C05403=1026.650,-101.229,-87.108,166.767,45.129,158.260
C05404=1026.657,-100.943,-87.119,166.771,45.126,158.259
C05405=1026.664,-100.656,-87.129,166.774,45.123,158.259
C05406=1026.670,-100.371,-87.141,166.778,45.121,158.259
C05407=1026.676,-100.120,-87.149,166.781,45.118,158.259
C05408=1026.681,-99.870,-87.160,166.783,45.115,158.259
C05409=1026.687,-99.621,-87.169,166.787,45.113,158.259
C05410=1026.693,-99.371,-87.178,166.789,45.110,158.259
C05411=1026.699,-99.122,-87.188,166.793,45.108,158.259
C05412=1026.705,-98.872,-87.198,166.795,45.105,158.258
C05413=1026.711,-98.622,-87.208,166.799,45.103,158.258
C05414=1026.716,-98.373,-87.217,166.801,45.101,158.258
C05415=1026.722,-98.123,-87.226,166.805,45.098,158.258
C05416=1026.729,-97.873,-87.236,166.807,45.096,158.258
C05417=1026.735,-97.623,-87.246,166.811,45.093,158.258
C05418=1026.740,-97.374,-87.255,166.813,45.091,158.258
C05419=1026.746,-97.124,-87.265,166.817,45.088,158.258
C05420=1026.751,-96.874,-87.275,166.819,45.086,158.257
C05421=1026.757,-96.624,-87.285,166.822,45.084,158.257
C05422=1026.763,-96.374,-87.295,166.825,45.081,158.257
C05423=1026.768,-96.125,-87.304,166.828,45.079,158.257
C05424=1026.774,-95.875,-87.314,166.831,45.077,158.257
C05425=1026.780,-95.625,-87.324,166.834,45.074,158.257
C05426=1026.786,-95.376,-87.335,166.837,45.072,158.257
C05427=1026.792,-95.126,-87.344,166.840,45.069,158.257
C05428=1026.797,-94.876,-87.354,166.843,45.067,158.257
C05429=1026.803,-94.627,-87.364,166.846,45.065,158.257
C05430=1026.808,-94.376,-87.374,166.848,45.062,158.256
C05431=1026.815,-94.127,-87.383,166.852,45.060,158.256
C05432=1026.820,-93.876,-87.393,166.854,45.058,158.256
C05433=1026.826,-93.627,-87.404,166.858,45.055,158.256
C05434=1026.831,-93.378,-87.414,166.860,45.053,158.256
C05435=1026.837,-93.128,-87.423,166.864,45.050,158.256
C05436=1026.843,-92.878,-87.433,166.866,45.048,158.256
C05437=1026.849,-92.628,-87.443,166.869,45.046,158.256
C05438=1026.855,-92.379,-87.454,166.872,45.043,158.255
C05439=1026.861,-92.129,-87.463,166.875,45.041,158.255
C05440=1026.866,-91.879,-87.473,166.878,45.038,158.255
C05441=1026.873,-91.629,-87.483,166.881,45.036,158.255
C05442=1026.878,-91.380,-87.494,166.884,45.033,158.255
C05443=1026.884,-91.130,-87.503,166.887,45.031,158.255
C05444=1026.889,-90.880,-87.513,166.891,45.029,158.255
C05445=1026.896,-90.631,-87.524,166.893,45.026,158.255
C05446=1026.901,-90.381,-87.534,166.895,45.024,158.255
C05447=1026.907,-90.131,-87.543,166.899,45.022,158.254
C05448=1026.913,-89.881,-87.553,166.901,45.020,158.254
C05449=1026.919,-89.632,-87.564,166.905,45.017,158.254
C05450=1026.925,-89.382,-87.574,166.907,45.015,158.254
C05451=1026.931,-89.132,-87.583,166.911,45.012,158.254
C05452=1026.937,-88.883,-87.594,166.913,45.010,158.254
C05453=1026.943,-88.633,-87.604,166.917,45.008,158.254
C05454=1026.948,-88.383,-87.614,166.919,45.005,158.254
C05455=1026.955,-88.133,-87.624,166.922,45.003,158.253
C05456=1026.960,-87.883,-87.634,166.926,45.001,158.253
C05457=1026.967,-87.634,-87.645,166.928,44.998,158.253
C05458=1026.972,-87.384,-87.655,166.932,44.996,158.253
C05459=1026.978,-87.134,-87.665,166.934,44.993,158.253
C05460=1026.984,-86.885,-87.675,166.937,44.991,158.253
C05461=1026.990,-86.635,-87.685,166.940,44.988,158.253
C05462=1026.996,-86.385,-87.696,166.943,44.986,158.253
C05463=1027.001,-86.135,-87.706,166.946,44.984,158.253
C05464=1027.008,-85.886,-87.716,166.948,44.981,158.252
C05465=1027.013,-85.636,-87.726,166.952,44.979,158.252
C05466=1027.019,-85.386,-87.736,166.954,44.976,158.252
C05467=1027.026,-85.103,-87.748,166.958,44.974,158.252
C05468=1027.033,-84.819,-87.760,166.961,44.971,158.252
C05469=1027.040,-84.534,-87.772,166.965,44.968,158.252
C05470=1027.046,-84.250,-87.783,166.968,44.966,158.252
C05471=1027.053,-84.001,-87.793,166.971,44.964,158.251
C05472=1027.058,-83.751,-87.804,166.974,44.961,158.251
C05473=1027.065,-83.502,-87.814,166.977,44.959,158.251
C05474=1027.070,-83.252,-87.824,166.980,44.956,158.251
C05475=1027.077,-83.002,-87.835,166.983,44.954,158.251
C05476=1027.083,-82.752,-87.845,166.986,44.952,158.251
C05477=1027.088,-82.502,-87.856,166.989,44.949,158.251
C05478=1027.094,-82.252,-87.865,166.992,44.947,158.251
C05479=1027.100,-82.003,-87.876,166.995,44.944,158.250
C05480=1027.107,-81.754,-87.886,166.997,44.942,158.250
C05481=1027.112,-81.503,-87.897,167.001,44.939,158.250
C05482=1027.119,-81.254,-87.907,167.003,44.937,158.250
C05483=1027.125,-81.003,-87.917,167.007,44.934,158.250
C05484=1027.130,-80.754,-87.928,167.009,44.932,158.250
C05485=1027.137,-80.505,-87.939,167.013,44.929,158.250
C05486=1027.142,-80.255,-87.949,167.015,44.927,158.250
C05487=1027.149,-80.006,-87.959,167.019,44.925,158.250
C05488=1027.154,-79.756,-87.970,167.021,44.922,158.249
C05489=1027.161,-79.505,-87.980,167.024,44.920,158.249
C05490=1027.166,-79.256,-87.991,167.027,44.918,158.249
C05491=1027.172,-79.006,-88.002,167.030,44.916,158.249
C05492=1027.178,-78.757,-88.012,167.032,44.914,158.249
C05493=1027.184,-78.507,-88.023,167.036,44.911,158.249
C05494=1027.190,-78.257,-88.034,167.038,44.909,158.249
C05495=1027.196,-78.007,-88.045,167.042,44.907,158.249
C05496=1027.202,-77.758,-88.056,167.044,44.905,158.248
C05497=1027.207,-77.508,-88.066,167.047,44.903,158.248
C05498=1027.214,-77.258,-88.076,167.050,44.900,158.248
C05499=1027.220,-77.008,-88.087,167.053,44.898,158.248
C05500=1027.226,-76.759,-88.098,167.056,44.896,158.248
C05501=1027.231,-76.509,-88.109,167.059,44.893,158.248
C05502=1027.237,-76.260,-88.120,167.062,44.891,158.248
C05503=1027.243,-76.010,-88.131,167.065,44.889,158.248
C05504=1027.250,-75.760,-88.141,167.068,44.887,158.248
C05505=1027.255,-75.510,-88.152,167.070,44.884,158.247
C05506=1027.261,-75.261,-88.162,167.074,44.882,158.247
C05507=1027.267,-75.011,-88.173,167.076,44.880,158.247
C05508=1027.273,-74.761,-88.185,167.079,44.877,158.247
C05509=1027.279,-74.512,-88.195,167.082,44.875,158.247
C05510=1027.285,-74.262,-88.206,167.085,44.873,158.247
C05511=1027.290,-74.013,-88.217,167.089,44.871,158.247
C05512=1027.297,-73.763,-88.228,167.091,44.868,158.247
C05513=1027.303,-73.513,-88.239,167.094,44.866,158.247
C05514=1027.308,-73.264,-88.250,167.096,44.864,158.246
C05515=1027.315,-73.013,-88.261,167.100,44.862,158.246
C05516=1027.320,-72.764,-88.272,167.102,44.860,158.246
C05517=1027.326,-72.514,-88.283,167.105,44.858,158.246
C05518=1027.331,-72.265,-88.295,167.109,44.856,158.246
C05519=1027.337,-72.014,-88.306,167.111,44.854,158.246
C05520=1027.343,-71.765,-88.317,167.113,44.851,158.246
C05521=1027.349,-71.515,-88.328,167.117,44.849,158.246
C05522=1027.355,-71.265,-88.339,167.120,44.847,158.246
C05523=1027.361,-71.016,-88.350,167.122,44.845,158.246
C05524=1027.367,-70.766,-88.361,167.125,44.843,158.246
C05525=1027.373,-70.517,-88.373,167.129,44.841,158.246
C05526=1027.378,-70.267,-88.384,167.131,44.839,158.245
C05527=1027.384,-70.017,-88.395,167.134,44.837,158.245
C05528=1027.390,-69.767,-88.406,167.137,44.834,158.245
C05529=1027.396,-69.518,-88.417,167.140,44.832,158.245
C05530=1027.402,-69.268,-88.428,167.142,44.830,158.245
C05531=1027.408,-68.987,-88.441,167.146,44.828,158.245
C05532=1027.416,-68.704,-88.454,167.149,44.825,158.245
///RCONF 1,0,0,1,0,0,0,0,0,0,0,0,0,0,0,0,0,0,0,0,0,0,0,0
C05533=1027.422,-68.423,-88.466,167.152,44.823,158.245
C05534=1027.428,-68.141,-88.479,167.155,44.820,158.245
C05535=1027.435,-67.891,-88.491,167.158,44.818,158.244
C05536=1027.441,-67.641,-88.502,167.161,44.816,158.244
C05537=1027.447,-67.391,-88.513,167.164,44.814,158.244
C05538=1027.453,-67.142,-88.524,167.167,44.812,158.244
C05539=1027.458,-66.892,-88.535,167.170,44.810,158.244
C05540=1027.464,-66.642,-88.547,167.173,44.807,158.244
C05541=1027.470,-66.393,-88.558,167.175,44.805,158.244
C05542=1027.476,-66.143,-88.570,167.178,44.803,158.244
C05543=1027.482,-65.894,-88.581,167.181,44.801,158.244
C05544=1027.488,-65.644,-88.592,167.184,44.799,158.244
C05545=1027.494,-65.394,-88.604,167.187,44.797,158.244
C05546=1027.499,-65.144,-88.615,167.190,44.794,158.243
C05547=1027.506,-64.895,-88.627,167.193,44.792,158.243
C05548=1027.512,-64.645,-88.638,167.195,44.790,158.243
C05549=1027.518,-64.395,-88.649,167.199,44.788,158.243
C05550=1027.524,-64.146,-88.660,167.201,44.786,158.243
C05551=1027.530,-63.896,-88.672,167.204,44.784,158.243
C05552=1027.536,-63.646,-88.683,167.206,44.781,158.243
C05553=1027.542,-63.397,-88.695,167.210,44.779,158.243
C05554=1027.548,-63.147,-88.706,167.213,44.777,158.243
C05555=1027.555,-62.898,-88.718,167.215,44.775,158.242
C05556=1027.560,-62.648,-88.729,167.219,44.773,158.242
C05557=1027.566,-62.398,-88.741,167.221,44.770,158.242
C05558=1027.572,-62.149,-88.752,167.224,44.768,158.242
C05559=1027.578,-61.899,-88.763,167.227,44.766,158.242
C05560=1027.584,-61.650,-88.775,167.230,44.764,158.242
C05561=1027.590,-61.399,-88.787,167.233,44.762,158.242
C05562=1027.596,-61.150,-88.798,167.235,44.760,158.242
C05563=1027.602,-60.900,-88.810,167.239,44.757,158.242
C05564=1027.608,-60.651,-88.821,167.241,44.755,158.241
C05565=1027.615,-60.401,-88.833,167.244,44.753,158.241
C05566=1027.620,-60.151,-88.844,167.247,44.751,158.241
C05567=1027.626,-59.902,-88.856,167.250,44.749,158.241
C05568=1027.633,-59.652,-88.867,167.252,44.747,158.241
C05569=1027.639,-59.403,-88.879,167.255,44.745,158.241
C05570=1027.645,-59.152,-88.890,167.259,44.742,158.241
C05571=1027.650,-58.903,-88.902,167.261,44.740,158.241
C05572=1027.657,-58.653,-88.914,167.264,44.738,158.241
C05573=1027.663,-58.404,-88.925,167.267,44.736,158.240
C05574=1027.669,-58.154,-88.936,167.270,44.734,158.240
C05575=1027.676,-57.904,-88.948,167.272,44.732,158.240
C05576=1027.681,-57.655,-88.960,167.276,44.729,158.240
C05577=1027.687,-57.405,-88.972,167.278,44.727,158.240
C05578=1027.694,-57.155,-88.983,167.281,44.725,158.240
C05579=1027.700,-56.906,-88.995,167.284,44.723,158.240
C05580=1027.706,-56.656,-89.007,167.287,44.721,158.240
C05581=1027.712,-56.407,-89.018,167.289,44.718,158.240
C05582=1027.718,-56.157,-89.030,167.292,44.716,158.239
C05583=1027.725,-55.907,-89.041,167.296,44.714,158.239
C05584=1027.731,-55.658,-89.053,167.298,44.712,158.239
C05585=1027.736,-55.408,-89.065,167.301,44.709,158.239
C05586=1027.743,-55.158,-89.077,167.303,44.707,158.239
C05587=1027.749,-54.909,-89.088,167.307,44.705,158.239
C05588=1027.756,-54.660,-89.100,167.309,44.703,158.239
C05589=1027.761,-54.409,-89.112,167.312,44.700,158.239
C05590=1027.768,-54.159,-89.124,167.315,44.698,158.239
C05591=1027.774,-53.911,-89.136,167.318,44.696,158.238
C05592=1027.780,-53.660,-89.147,167.321,44.694,158.238
C05593=1027.786,-53.410,-89.159,167.324,44.692,158.238
C05594=1027.792,-53.162,-89.171,167.327,44.690,158.238
C05595=1027.799,-52.881,-89.184,167.329,44.687,158.238
C05596=1027.806,-52.600,-89.198,167.333,44.685,158.238
C05597=1027.813,-52.319,-89.210,167.336,44.682,158.238
C05598=1027.821,-52.038,-89.224,167.340,44.680,158.238
C05599=1027.826,-51.788,-89.236,167.342,44.678,158.237
C05600=1027.832,-51.539,-89.247,167.345,44.675,158.237
C05601=1027.839,-51.290,-89.259,167.347,44.673,158.237
C05602=1027.846,-51.040,-89.271,167.351,44.671,158.237
C05603=1027.851,-50.789,-89.283,167.353,44.668,158.237
C05604=1027.858,-50.540,-89.295,167.356,44.666,158.237
C05605=1027.863,-50.291,-89.307,167.358,44.664,158.237
C05606=1027.869,-50.041,-89.320,167.362,44.662,158.237
C05607=1027.876,-49.791,-89.332,167.365,44.660,158.236
C05608=1027.882,-49.541,-89.344,167.367,44.658,158.236
C05609=1027.888,-49.293,-89.356,167.370,44.656,158.236
C05610=1027.894,-49.043,-89.369,167.372,44.654,158.236
C05611=1027.900,-48.793,-89.381,167.376,44.652,158.236
C05612=1027.906,-48.543,-89.393,167.379,44.650,158.236
C05613=1027.912,-48.294,-89.405,167.381,44.648,158.236
C05614=1027.917,-48.044,-89.418,167.384,44.646,158.236
C05615=1027.924,-47.795,-89.430,167.386,44.644,158.236
C05616=1027.930,-47.545,-89.442,167.389,44.642,158.236
C05617=1027.937,-47.295,-89.454,167.393,44.640,158.236
C05618=1027.942,-47.046,-89.466,167.395,44.638,158.235
C05619=1027.948,-46.796,-89.479,167.398,44.636,158.235
C05620=1027.954,-46.546,-89.491,167.400,44.634,158.235
C05621=1027.960,-46.297,-89.503,167.403,44.632,158.235
C05622=1027.966,-46.047,-89.516,167.407,44.630,158.235
C05623=1027.972,-45.798,-89.528,167.409,44.628,158.235
C05624=1027.978,-45.548,-89.540,167.412,44.626,158.235
C05625=1027.984,-45.298,-89.553,167.414,44.624,158.235
C05626=1027.991,-45.048,-89.565,167.417,44.622,158.235
C05627=1027.997,-44.799,-89.577,167.420,44.619,158.235
C05628=1028.003,-44.549,-89.590,167.423,44.617,158.234
C05629=1028.009,-44.300,-89.601,167.426,44.615,158.234
C05630=1028.015,-44.050,-89.614,167.428,44.614,158.234
C05631=1028.020,-43.800,-89.627,167.431,44.612,158.234
C05632=1028.027,-43.551,-89.639,167.433,44.610,158.234
C05633=1028.033,-43.301,-89.652,167.437,44.607,158.234
C05634=1028.039,-43.051,-89.664,167.440,44.605,158.234
C05635=1028.046,-42.802,-89.676,167.442,44.604,158.234
C05636=1028.052,-42.552,-89.689,167.445,44.602,158.234
C05637=1028.058,-42.302,-89.701,167.447,44.600,158.234
C05638=1028.064,-42.052,-89.713,167.451,44.597,158.233
C05639=1028.070,-41.804,-89.726,167.453,44.595,158.233
C05640=1028.076,-41.554,-89.739,167.456,44.593,158.233
C05641=1028.083,-41.304,-89.751,167.459,44.591,158.233
C05642=1028.088,-41.055,-89.763,167.461,44.589,158.233
C05643=1028.094,-40.805,-89.776,167.464,44.587,158.233
C05644=1028.101,-40.556,-89.789,167.467,44.585,158.233
C05645=1028.107,-40.306,-89.801,167.470,44.583,158.233
C05646=1028.113,-40.056,-89.814,167.473,44.581,158.233
C05647=1028.120,-39.806,-89.826,167.475,44.579,158.232
C05648=1028.126,-39.557,-89.839,167.478,44.576,158.232
C05649=1028.132,-39.307,-89.851,167.481,44.574,158.232
C05650=1028.139,-39.058,-89.863,167.484,44.572,158.232
C05651=1028.144,-38.808,-89.876,167.486,44.570,158.232
C05652=1028.151,-38.558,-89.889,167.489,44.568,158.232
C05653=1028.157,-38.309,-89.902,167.492,44.566,158.232
C05654=1028.162,-38.059,-89.914,167.494,44.564,158.232
C05655=1028.169,-37.809,-89.928,167.497,44.562,158.232
C05656=1028.175,-37.560,-89.940,167.499,44.560,158.231
C05657=1028.181,-37.310,-89.953,167.503,44.558,158.231
C05658=1028.187,-37.060,-89.966,167.506,44.557,158.231
C05659=1028.194,-36.780,-89.981,167.508,44.554,158.231
C05660=1028.200,-36.500,-89.994,167.512,44.552,158.231
C05661=1028.207,-36.220,-90.009,167.514,44.550,158.231
C05662=1028.214,-35.940,-90.023,167.518,44.548,158.231
C05663=1028.220,-35.690,-90.037,167.521,44.546,158.231
C05664=1028.226,-35.440,-90.049,167.523,44.544,158.231
C05665=1028.232,-35.191,-90.062,167.526,44.542,158.231
C05666=1028.238,-34.941,-90.075,167.528,44.540,158.231
C05667=1028.244,-34.691,-90.087,167.531,44.538,158.230
C05668=1028.250,-34.442,-90.101,167.534,44.536,158.230
C05669=1028.257,-34.193,-90.113,167.536,44.534,158.230
C05670=1028.263,-33.943,-90.126,167.539,44.532,158.230
C05671=1028.269,-33.693,-90.139,167.542,44.530,158.230
C05672=1028.276,-33.443,-90.152,167.545,44.528,158.230
C05673=1028.282,-33.194,-90.165,167.548,44.526,158.230
C05674=1028.288,-32.944,-90.178,167.550,44.524,158.230
C05675=1028.294,-32.695,-90.191,167.553,44.522,158.230
C05676=1028.300,-32.445,-90.204,167.555,44.520,158.230
C05677=1028.306,-32.196,-90.217,167.558,44.519,158.229
C05678=1028.312,-31.946,-90.230,167.561,44.517,158.229
C05679=1028.318,-31.697,-90.243,167.563,44.515,158.229
C05680=1028.324,-31.447,-90.255,167.567,44.512,158.229
C05681=1028.330,-31.198,-90.269,167.570,44.511,158.229
C05682=1028.337,-30.948,-90.282,167.572,44.509,158.229
C05683=1028.343,-30.698,-90.295,167.575,44.507,158.229
C05684=1028.349,-30.448,-90.308,167.577,44.505,158.229
C05685=1028.356,-30.199,-90.321,167.580,44.502,158.228
C05686=1028.361,-29.949,-90.334,167.582,44.500,158.228
C05687=1028.368,-29.700,-90.347,167.585,44.498,158.228
C05688=1028.374,-29.450,-90.360,167.587,44.496,158.228
///RCONF 1,0,0,0,0,0,0,0,0,0,0,0,0,0,0,0,0,0,0,0,0,0,0,0
C05689=1028.380,-29.201,-90.373,167.591,44.494,158.228
C05690=1028.387,-28.951,-90.387,167.594,44.492,158.228
C05691=1028.393,-28.701,-90.399,167.596,44.490,158.228
C05692=1028.399,-28.452,-90.413,167.599,44.488,158.228
C05693=1028.405,-28.203,-90.426,167.602,44.486,158.228
C05694=1028.411,-27.953,-90.438,167.604,44.484,158.228
C05695=1028.418,-27.703,-90.452,167.607,44.482,158.227
C05696=1028.424,-27.453,-90.465,167.609,44.480,158.227
C05697=1028.430,-27.204,-90.479,167.612,44.478,158.227
C05698=1028.436,-26.954,-90.491,167.615,44.476,158.227
C05699=1028.442,-26.705,-90.504,167.617,44.475,158.227
C05700=1028.448,-26.456,-90.518,167.620,44.473,158.227
C05701=1028.455,-26.205,-90.532,167.623,44.470,158.227
C05702=1028.461,-25.956,-90.545,167.626,44.468,158.227
C05703=1028.467,-25.707,-90.558,167.629,44.467,158.227
C05704=1028.473,-25.457,-90.571,167.631,44.465,158.227
C05705=1028.478,-25.207,-90.585,167.634,44.463,158.227
C05706=1028.485,-24.958,-90.598,167.637,44.461,158.226
C05707=1028.491,-24.708,-90.612,167.639,44.459,158.226
C05708=1028.498,-24.459,-90.625,167.642,44.457,158.226
C05709=1028.503,-24.209,-90.639,167.644,44.456,158.226
C05710=1028.509,-23.960,-90.652,167.647,44.454,158.226
C05711=1028.516,-23.710,-90.666,167.650,44.452,158.226
C05712=1028.522,-23.460,-90.678,167.652,44.450,158.226
C05713=1028.527,-23.211,-90.692,167.655,44.448,158.226
C05714=1028.534,-22.961,-90.705,167.657,44.446,158.226
C05715=1028.540,-22.718,-90.719,167.660,44.445,158.226
C05716=1028.546,-22.474,-90.732,167.663,44.443,158.226
C05717=1028.552,-22.230,-90.745,167.665,44.441,158.225
C05718=1028.558,-21.987,-90.759,167.668,44.439,158.225
C05719=1028.564,-21.743,-90.772,167.671,44.437,158.225
C05720=1028.570,-21.499,-90.785,167.673,44.435,158.225
C05721=1028.576,-21.255,-90.799,167.676,44.433,158.225
C05722=1028.582,-21.011,-90.811,167.678,44.431,158.225
C05723=1028.590,-20.718,-90.827,167.681,44.429,158.225
C05724=1028.597,-20.426,-90.843,167.685,44.427,158.225
C05725=1028.605,-20.133,-90.859,167.687,44.424,158.224
C05726=1028.611,-19.841,-90.875,167.691,44.422,158.224
C05727=1028.618,-19.591,-90.889,167.693,44.420,158.224
C05728=1028.624,-19.341,-90.902,167.696,44.418,158.224
C05729=1028.630,-19.092,-90.916,167.698,44.416,158.224
C05730=1028.637,-18.842,-90.930,167.701,44.414,158.224
C05731=1028.643,-18.593,-90.943,167.704,44.412,158.224
C05732=1028.648,-18.343,-90.957,167.706,44.410,158.224
C05733=1028.655,-18.093,-90.970,167.709,44.408,158.224
C05734=1028.661,-17.844,-90.984,167.711,44.406,158.223
C05735=1028.668,-17.594,-90.997,167.714,44.405,158.223
C05736=1028.674,-17.344,-91.011,167.717,44.403,158.223
C05737=1028.680,-17.095,-91.024,167.719,44.401,158.223
C05738=1028.686,-16.846,-91.038,167.722,44.399,158.223
C05739=1028.692,-16.596,-91.053,167.724,44.397,158.223
C05740=1028.699,-16.347,-91.066,167.727,44.395,158.223
C05741=1028.705,-16.097,-91.080,167.730,44.393,158.223
C05742=1028.711,-15.847,-91.093,167.732,44.391,158.223
C05743=1028.717,-15.598,-91.107,167.735,44.389,158.222
C05744=1028.724,-15.348,-91.120,167.737,44.387,158.222
C05745=1028.730,-15.099,-91.135,167.740,44.385,158.222
C05746=1028.737,-14.849,-91.149,167.743,44.384,158.222
C05747=1028.742,-14.599,-91.162,167.746,44.382,158.222
C05748=1028.747,-14.350,-91.176,167.748,44.380,158.222
C05749=1028.755,-14.101,-91.191,167.751,44.378,158.222
C05750=1028.760,-13.851,-91.204,167.753,44.376,158.222
C05751=1028.767,-13.601,-91.218,167.756,44.374,158.222
C05752=1028.772,-13.351,-91.232,167.759,44.372,158.222
C05753=1028.779,-13.103,-91.246,167.761,44.370,158.221
C05754=1028.785,-12.853,-91.260,167.764,44.369,158.222
C05755=1028.791,-12.603,-91.273,167.767,44.367,158.221
C05756=1028.798,-12.354,-91.288,167.769,44.365,158.221
C05757=1028.803,-12.104,-91.302,167.772,44.363,158.221
C05758=1028.810,-11.854,-91.316,167.774,44.361,158.221
C05759=1028.816,-11.605,-91.330,167.777,44.359,158.221
C05760=1028.822,-11.356,-91.344,167.780,44.357,158.221
C05761=1028.828,-11.106,-91.359,167.782,44.355,158.221
C05762=1028.834,-10.857,-91.372,167.785,44.353,158.221
C05763=1028.841,-10.607,-91.386,167.788,44.352,158.221
C05764=1028.847,-10.358,-91.400,167.790,44.350,158.221
C05765=1028.853,-10.108,-91.414,167.793,44.348,158.220
C05766=1028.859,-9.858,-91.428,167.795,44.346,158.220
C05767=1028.866,-9.609,-91.443,167.798,44.344,158.220
C05768=1028.871,-9.359,-91.456,167.801,44.343,158.220
C05769=1028.878,-9.110,-91.471,167.803,44.341,158.220
C05770=1028.884,-8.860,-91.485,167.806,44.339,158.220
C05771=1028.891,-8.611,-91.499,167.808,44.337,158.220
C05772=1028.896,-8.361,-91.513,167.811,44.335,158.220
C05773=1028.903,-8.112,-91.528,167.813,44.333,158.219
C05774=1028.909,-7.862,-91.541,167.815,44.331,158.219
C05775=1028.915,-7.612,-91.555,167.818,44.329,158.219
C05776=1028.922,-7.364,-91.569,167.821,44.328,158.219
C05777=1028.928,-7.113,-91.584,167.823,44.326,158.219
C05778=1028.933,-6.864,-91.598,167.826,44.324,158.219
C05779=1028.940,-6.614,-91.612,167.828,44.322,158.219
C05780=1028.947,-6.365,-91.627,167.831,44.320,158.219
C05781=1028.953,-6.115,-91.640,167.834,44.318,158.219
C05782=1028.959,-5.866,-91.655,167.836,44.316,158.219
C05783=1028.965,-5.616,-91.669,167.839,44.314,158.218
C05784=1028.972,-5.367,-91.683,167.841,44.312,158.218
C05785=1028.978,-5.118,-91.698,167.844,44.310,158.218
C05786=1028.984,-4.868,-91.711,167.847,44.309,158.218
C05787=1028.991,-4.585,-91.727,167.849,44.307,158.218
C05788=1028.998,-4.302,-91.744,167.853,44.304,158.218
C05789=1029.006,-4.020,-91.760,167.855,44.302,158.218
C05790=1029.013,-3.736,-91.776,167.858,44.300,158.218
C05791=1029.018,-3.487,-91.791,167.861,44.298,158.217
C05792=1029.025,-3.238,-91.806,167.863,44.297,158.217
C05793=1029.031,-2.988,-91.821,167.866,44.295,158.217
C05794=1029.037,-2.739,-91.835,167.869,44.293,158.217
C05795=1029.043,-2.489,-91.849,167.871,44.291,158.217
C05796=1029.049,-2.240,-91.864,167.874,44.289,158.217
C05797=1029.056,-1.991,-91.878,167.877,44.288,158.217
C05798=1029.061,-1.741,-91.892,167.878,44.286,158.217
C05799=1029.068,-1.491,-91.907,167.881,44.284,158.217
C05800=1029.074,-1.242,-91.922,167.883,44.282,158.217
C05801=1029.080,-0.993,-91.937,167.886,44.281,158.217
C05802=1029.086,-0.742,-91.951,167.889,44.279,158.216
C05803=1029.092,-0.494,-91.966,167.891,44.277,158.216
C05804=1029.098,-0.244,-91.980,167.894,44.275,158.216
C05805=1029.105,0.006,-91.995,167.897,44.273,158.216
C05806=1029.110,0.255,-92.010,167.898,44.271,158.216
C05807=1029.116,0.505,-92.024,167.901,44.270,158.216
C05808=1029.123,0.755,-92.039,167.904,44.268,158.216
C05809=1029.129,1.004,-92.054,167.906,44.266,158.216
C05810=1029.135,1.253,-92.069,167.909,44.264,158.216
C05811=1029.141,1.503,-92.084,167.911,44.262,158.216
C05812=1029.147,1.752,-92.098,167.914,44.261,158.216
C05813=1029.153,2.002,-92.112,167.917,44.259,158.215
C05814=1029.160,2.252,-92.127,167.918,44.258,158.215
C05815=1029.166,2.500,-92.141,167.921,44.256,158.215
C05816=1029.173,2.750,-92.156,167.924,44.254,158.215
C05817=1029.179,3.000,-92.171,167.926,44.252,158.215
C05818=1029.185,3.249,-92.186,167.929,44.251,158.215
C05819=1029.191,3.498,-92.201,167.932,44.249,158.215
C05820=1029.197,3.748,-92.216,167.934,44.247,158.215
C05821=1029.203,3.997,-92.230,167.937,44.245,158.215
C05822=1029.210,4.247,-92.245,167.939,44.243,158.214
C05823=1029.216,4.496,-92.260,167.941,44.241,158.214
C05824=1029.221,4.746,-92.274,167.944,44.239,158.214
C05825=1029.228,4.996,-92.289,167.947,44.238,158.214
C05826=1029.234,5.245,-92.304,167.949,44.236,158.214
C05827=1029.241,5.495,-92.319,167.952,44.234,158.214
C05828=1029.246,5.744,-92.334,167.954,44.232,158.214
C05829=1029.253,5.993,-92.348,167.957,44.230,158.214
C05830=1029.259,6.243,-92.363,167.960,44.228,158.214
C05831=1029.266,6.493,-92.378,167.961,44.227,158.213
C05832=1029.271,6.742,-92.393,167.964,44.225,158.213
C05833=1029.278,6.991,-92.408,167.966,44.223,158.213
C05834=1029.284,7.241,-92.423,167.969,44.221,158.213
C05835=1029.290,7.491,-92.438,167.972,44.220,158.213
C05836=1029.297,7.740,-92.453,167.974,44.218,158.213
C05837=1029.303,7.989,-92.467,167.977,44.216,158.213
C05838=1029.309,8.239,-92.482,167.980,44.214,158.213
C05839=1029.315,8.489,-92.497,167.981,44.212,158.213
C05840=1029.322,8.738,-92.513,167.984,44.210,158.212
C05841=1029.328,8.987,-92.528,167.986,44.208,158.212
C05842=1029.334,9.236,-92.542,167.989,44.206,158.212
C05843=1029.341,9.486,-92.557,167.992,44.204,158.212
C05844=1029.347,9.736,-92.572,167.994,44.202,158.212
C05845=1029.353,9.985,-92.587,167.997,44.200,158.212
C05846=1029.360,10.235,-92.602,167.999,44.199,158.212
C05847=1029.366,10.484,-92.617,168.002,44.197,158.212
C05848=1029.372,10.734,-92.632,168.004,44.196,158.212
C05849=1029.378,10.983,-92.647,168.006,44.194,158.211
C05850=1029.385,11.232,-92.662,168.009,44.192,158.211
C05851=1029.392,11.517,-92.679,168.011,44.189,158.211
C05852=1029.399,11.802,-92.696,168.015,44.187,158.211
C05853=1029.407,12.087,-92.713,168.018,44.185,158.211
C05854=1029.414,12.371,-92.731,168.020,44.183,158.211
C05855=1029.420,12.621,-92.746,168.023,44.181,158.211
C05856=1029.427,12.871,-92.760,168.025,44.179,158.210
C05857=1029.433,13.120,-92.775,168.028,44.177,158.210
C05858=1029.440,13.369,-92.791,168.031,44.175,158.210
C05859=1029.445,13.618,-92.806,168.033,44.174,158.210
C05860=1029.452,13.868,-92.821,168.036,44.172,158.210
C05861=1029.458,14.118,-92.836,168.037,44.170,158.210
C05862=1029.464,14.367,-92.852,168.040,44.168,158.210
C05863=1029.471,14.617,-92.867,168.043,44.166,158.210
C05864=1029.477,14.866,-92.882,168.046,44.165,158.210
C05865=1029.484,15.115,-92.897,168.048,44.163,158.209
C05866=1029.489,15.365,-92.913,168.051,44.161,158.209
C05867=1029.496,15.615,-92.928,168.052,44.159,158.209
C05868=1029.502,15.863,-92.943,168.055,44.157,158.209
C05869=1029.508,16.113,-92.958,168.058,44.155,158.209
C05870=1029.514,16.363,-92.974,168.060,44.154,158.209
C05871=1029.520,16.612,-92.989,168.063,44.152,158.209
C05872=1029.527,16.862,-93.004,168.065,44.151,158.209
C05873=1029.532,17.112,-93.020,168.067,44.149,158.209
C05874=1029.539,17.361,-93.035,168.070,44.147,158.208
C05875=1029.546,17.610,-93.050,168.072,44.145,158.208
C05876=1029.552,17.859,-93.066,168.075,44.143,158.208
C05877=1029.558,18.109,-93.082,168.078,44.142,158.208
C05878=1029.564,18.359,-93.097,168.079,44.140,158.208
C05879=1029.571,18.608,-93.112,168.082,44.138,158.208
C05880=1029.577,18.858,-93.128,168.085,44.136,158.208
C05881=1029.583,19.107,-93.143,168.087,44.134,158.208
C05882=1029.589,19.356,-93.158,168.090,44.132,158.208
C05883=1029.596,19.605,-93.174,168.091,44.130,158.207
C05884=1029.601,19.855,-93.189,168.094,44.129,158.207
C05885=1029.608,20.104,-93.205,168.097,44.127,158.207
C05886=1029.614,20.354,-93.220,168.099,44.125,158.207
C05887=1029.620,20.603,-93.236,168.102,44.123,158.207
C05888=1029.626,20.853,-93.252,168.104,44.122,158.207
C05889=1029.633,21.102,-93.267,168.106,44.121,158.207
C05890=1029.639,21.352,-93.282,168.109,44.119,158.207
C05891=1029.645,21.601,-93.298,168.112,44.117,158.207
C05892=1029.651,21.851,-93.313,168.114,44.115,158.206
C05893=1029.657,22.100,-93.330,168.116,44.113,158.206
C05894=1029.664,22.350,-93.345,168.119,44.111,158.206
C05895=1029.670,22.599,-93.361,168.121,44.110,158.206
C05896=1029.676,22.848,-93.377,168.124,44.108,158.206
C05897=1029.682,23.098,-93.392,168.127,44.106,158.206
C05898=1029.689,23.347,-93.408,168.128,44.104,158.206
C05899=1029.695,23.597,-93.423,168.131,44.102,158.206
C05900=1029.701,23.846,-93.439,168.133,44.100,158.206
C05901=1029.708,24.095,-93.455,168.136,44.099,158.206
C05902=1029.713,24.345,-93.470,168.139,44.097,158.205
C05903=1029.720,24.594,-93.486,168.140,44.096,158.205
C05904=1029.726,24.843,-93.502,168.143,44.094,158.205
C05905=1029.732,25.093,-93.517,168.146,44.092,158.205
C05906=1029.739,25.343,-93.534,168.148,44.090,158.205
C05907=1029.746,25.592,-93.549,168.151,44.088,158.205
C05908=1029.752,25.842,-93.564,168.152,44.086,158.205
C05909=1029.758,26.091,-93.580,168.155,44.085,158.205
C05910=1029.765,26.340,-93.596,168.158,44.083,158.204
C05911=1029.770,26.590,-93.612,168.160,44.081,158.204
C05912=1029.777,26.839,-93.627,168.162,44.079,158.204
C05913=1029.783,27.089,-93.644,168.165,44.078,158.204
C05914=1029.789,27.338,-93.660,168.167,44.076,158.204
C05915=1029.797,27.624,-93.677,168.170,44.074,158.204
C05916=1029.804,27.910,-93.695,168.172,44.072,158.204
C05917=1029.811,28.196,-93.714,168.176,44.070,158.204
C05918=1029.818,28.482,-93.732,168.179,44.068,158.203
C05919=1029.823,28.732,-93.748,168.181,44.066,158.203
C05920=1029.830,28.981,-93.764,168.183,44.064,158.203
C05921=1029.836,29.230,-93.780,168.186,44.063,158.203
C05922=1029.842,29.479,-93.796,168.188,44.061,158.203
C05923=1029.849,29.729,-93.812,168.191,44.059,158.203
C05924=1029.855,29.979,-93.828,168.193,44.057,158.203
C05925=1029.861,30.228,-93.845,168.195,44.056,158.203
C05926=1029.868,30.478,-93.860,168.198,44.054,158.203
C05927=1029.874,30.727,-93.876,168.201,44.052,158.202
C05928=1029.879,30.976,-93.892,168.202,44.051,158.202
C05929=1029.886,31.225,-93.908,168.205,44.049,158.202
C05930=1029.892,31.475,-93.924,168.208,44.047,158.202
C05931=1029.899,31.725,-93.941,168.210,44.046,158.202
C05932=1029.905,31.974,-93.956,168.212,44.044,158.202
C05933=1029.911,32.223,-93.973,168.214,44.042,158.202
C05934=1029.917,32.472,-93.989,168.217,44.040,158.202
C05935=1029.923,32.722,-94.005,168.220,44.039,158.202
C05936=1029.930,32.971,-94.021,168.221,44.037,158.201
C05937=1029.936,33.221,-94.036,168.224,44.035,158.201
C05938=1029.942,33.471,-94.053,168.227,44.033,158.201
C05939=1029.949,33.720,-94.069,168.229,44.031,158.201
C05940=1029.955,33.969,-94.085,168.231,44.030,158.201
C05941=1029.961,34.219,-94.101,168.234,44.028,158.201
C05942=1029.967,34.468,-94.117,168.236,44.026,158.201
C05943=1029.973,34.717,-94.133,168.239,44.025,158.201
C05944=1029.980,34.967,-94.150,168.240,44.023,158.201
C05945=1029.986,35.216,-94.166,168.243,44.021,158.200
C05946=1029.993,35.465,-94.182,168.246,44.019,158.200
C05947=1029.998,35.715,-94.198,168.248,44.017,158.200
C05948=1030.005,35.965,-94.214,168.250,44.016,158.200
C05949=1030.012,36.214,-94.230,168.253,44.014,158.200
C05950=1030.018,36.463,-94.246,168.255,44.012,158.200
C05951=1030.024,36.712,-94.263,168.258,44.010,158.200
C05952=1030.030,36.961,-94.280,168.260,44.009,158.200
C05953=1030.037,37.211,-94.296,168.262,44.007,158.199
C05954=1030.043,37.460,-94.312,168.265,44.006,158.199
C05955=1030.049,37.710,-94.328,168.268,44.004,158.199
C05956=1030.055,37.959,-94.344,168.269,44.002,158.199
C05957=1030.062,38.209,-94.361,168.272,44.000,158.199
C05958=1030.068,38.458,-94.377,168.275,43.999,158.199
C05959=1030.074,38.707,-94.394,168.276,43.997,158.199
C05960=1030.080,38.956,-94.410,168.279,43.995,158.199
C05961=1030.086,39.206,-94.427,168.281,43.993,158.199
C05962=1030.092,39.456,-94.443,168.284,43.992,158.199
C05963=1030.098,39.705,-94.460,168.286,43.990,158.198
C05964=1030.104,39.955,-94.476,168.288,43.988,158.198
C05965=1030.110,40.203,-94.493,168.291,43.986,158.198
C05966=1030.117,40.453,-94.509,168.294,43.985,158.198
C05967=1030.123,40.703,-94.526,168.295,43.984,158.198
C05968=1030.129,40.952,-94.542,168.298,43.982,158.198
C05969=1030.135,41.201,-94.559,168.301,43.980,158.198
C05970=1030.142,41.451,-94.576,168.302,43.978,158.198
C05971=1030.148,41.700,-94.592,168.305,43.977,158.198
C05972=1030.154,41.950,-94.608,168.308,43.975,158.197
C05973=1030.161,42.199,-94.625,168.310,43.973,158.197
C05974=1030.167,42.448,-94.641,168.312,43.971,158.197
C05975=1030.173,42.697,-94.657,168.315,43.969,158.197
C05976=1030.179,42.946,-94.674,168.317,43.968,158.197
C05977=1030.185,43.196,-94.692,168.319,43.966,158.197
C05978=1030.191,43.446,-94.708,168.322,43.965,158.197
C05979=1030.199,43.731,-94.727,168.324,43.963,158.197
C05980=1030.205,44.018,-94.746,168.327,43.961,158.197
C05981=1030.212,44.303,-94.766,168.330,43.959,158.196
C05982=1030.219,44.589,-94.785,168.332,43.958,158.196
C05983=1030.225,44.838,-94.802,168.335,43.956,158.196
C05984=1030.231,45.089,-94.819,168.337,43.954,158.196
C05985=1030.237,45.338,-94.835,168.339,43.953,158.196
C05986=1030.243,45.587,-94.852,168.342,43.951,158.196
C05987=1030.250,45.837,-94.869,168.344,43.949,158.196
C05988=1030.256,46.086,-94.886,168.346,43.948,158.196
C05989=1030.262,46.335,-94.902,168.349,43.946,158.196
C05990=1030.268,46.584,-94.920,168.352,43.944,158.195
C05991=1030.274,46.834,-94.936,168.353,43.943,158.195
C05992=1030.281,47.083,-94.953,168.356,43.941,158.195
C05993=1030.286,47.333,-94.970,168.359,43.939,158.195
C05994=1030.293,47.582,-94.987,168.360,43.938,158.195
C05995=1030.299,47.831,-95.003,168.363,43.936,158.195
C05996=1030.305,48.080,-95.021,168.366,43.934,158.195
C05997=1030.311,48.330,-95.038,168.367,43.933,158.195
C05998=1030.317,48.579,-95.055,168.370,43.931,158.195
C05999=1030.323,48.829,-95.071,168.373,43.930,158.195
C06000=1030.330,49.078,-95.088,168.374,43.928,158.194
C06001=1030.335,49.327,-95.105,168.377,43.927,158.194
C06002=1030.342,49.577,-95.122,168.380,43.925,158.194
C06003=1030.348,49.826,-95.139,168.381,43.923,158.194
C06004=1030.355,50.075,-95.156,168.384,43.922,158.194
C06005=1030.360,50.324,-95.174,168.387,43.920,158.194
C06006=1030.366,50.574,-95.190,168.389,43.918,158.194
C06007=1030.373,50.823,-95.207,168.391,43.916,158.194
C06008=1030.379,51.073,-95.223,168.394,43.915,158.194
C06009=1030.385,51.322,-95.241,168.396,43.913,158.194
C06010=1030.391,51.571,-95.258,168.398,43.911,158.193
C06011=1030.397,51.820,-95.275,168.401,43.910,158.193
C06012=1030.404,52.070,-95.292,168.403,43.908,158.193
C06013=1030.409,52.320,-95.309,168.405,43.907,158.193
C06014=1030.416,52.569,-95.326,168.408,43.905,158.193
C06015=1030.422,52.818,-95.343,168.410,43.903,158.193
C06016=1030.429,53.068,-95.360,168.412,43.902,158.193
C06017=1030.434,53.317,-95.377,168.415,43.900,158.193
C06018=1030.441,53.565,-95.394,168.417,43.898,158.192
C06019=1030.447,53.816,-95.411,168.420,43.896,158.192
C06020=1030.453,54.065,-95.428,168.421,43.894,158.192
C06021=1030.460,54.314,-95.446,168.424,43.893,158.192
C06022=1030.466,54.563,-95.462,168.427,43.891,158.192
C06023=1030.472,54.813,-95.479,168.428,43.890,158.192
C06024=1030.478,55.062,-95.497,168.431,43.888,158.192
C06025=1030.485,55.311,-95.514,168.434,43.886,158.192
C06026=1030.491,55.561,-95.531,168.435,43.885,158.192
C06027=1030.498,55.810,-95.548,168.438,43.883,158.191
C06028=1030.503,56.059,-95.565,168.441,43.881,158.191
C06029=1030.510,56.309,-95.582,168.443,43.879,158.191
C06030=1030.516,56.558,-95.599,168.445,43.877,158.191
C06031=1030.522,56.808,-95.617,168.448,43.876,158.191
C06032=1030.528,57.056,-95.634,168.450,43.874,158.191
C06033=1030.535,57.306,-95.651,168.452,43.873,158.191
C06034=1030.541,57.555,-95.668,168.455,43.871,158.190
C06035=1030.547,57.805,-95.685,168.457,43.869,158.190
C06036=1030.554,58.054,-95.702,168.460,43.868,158.190
C06037=1030.560,58.303,-95.720,168.462,43.866,158.190
C06038=1030.566,58.553,-95.737,168.464,43.864,158.190
C06039=1030.572,58.802,-95.754,168.467,43.862,158.190
C06040=1030.579,59.052,-95.771,168.468,43.860,158.190
C06041=1030.586,59.300,-95.788,168.471,43.858,158.190
C06042=1030.592,59.550,-95.806,168.474,43.857,158.189
C06043=1030.599,59.836,-95.826,168.476,43.855,158.189
C06044=1030.606,60.122,-95.846,168.479,43.853,158.189
C06045=1030.613,60.406,-95.865,168.481,43.851,158.189
C06046=1030.620,60.692,-95.884,168.484,43.849,158.189
C06047=1030.627,60.942,-95.902,168.487,43.847,158.189
C06048=1030.633,61.192,-95.920,168.489,43.845,158.189
C06049=1030.640,61.440,-95.937,168.491,43.844,158.188
C06050=1030.647,61.690,-95.954,168.493,43.842,158.188
C06051=1030.652,61.939,-95.972,168.496,43.840,158.188
C06052=1030.659,62.189,-95.988,168.499,43.839,158.188
C06053=1030.665,62.438,-96.006,168.500,43.837,158.188
C06054=1030.672,62.687,-96.023,168.503,43.835,158.188
C06055=1030.678,62.937,-96.040,168.506,43.833,158.188
C06056=1030.684,63.185,-96.057,168.508,43.831,158.188
C06057=1030.691,63.435,-96.075,168.510,43.830,158.187
C06058=1030.697,63.685,-96.093,168.513,43.828,158.187
C06059=1030.703,63.934,-96.110,168.515,43.826,158.187
C06060=1030.709,64.183,-96.128,168.517,43.825,158.187
C06061=1030.716,64.433,-96.146,168.520,43.823,158.187
C06062=1030.722,64.682,-96.163,168.522,43.822,158.187
C06063=1030.728,64.931,-96.180,168.524,43.820,158.187
C06064=1030.734,65.180,-96.197,168.527,43.818,158.187
C06065=1030.740,65.430,-96.215,168.529,43.816,158.187
C06066=1030.746,65.679,-96.233,168.531,43.815,158.187
C06067=1030.753,65.928,-96.251,168.534,43.813,158.186
C06068=1030.759,66.177,-96.269,168.536,43.811,158.186
C06069=1030.766,66.427,-96.286,168.538,43.810,158.186
C06070=1030.772,66.676,-96.304,168.541,43.808,158.186
C06071=1030.778,66.926,-96.322,168.543,43.807,158.186
C06072=1030.784,67.174,-96.339,168.545,43.805,158.186
C06073=1030.790,67.424,-96.357,168.548,43.803,158.186
C06074=1030.796,67.674,-96.375,168.550,43.802,158.186
C06075=1030.803,67.922,-96.392,168.553,43.800,158.185
C06076=1030.809,68.172,-96.410,168.555,43.798,158.185
C06077=1030.815,68.421,-96.428,168.557,43.796,158.185
C06078=1030.821,68.670,-96.445,168.560,43.795,158.185
C06079=1030.827,68.920,-96.463,168.562,43.793,158.185
C06080=1030.834,69.169,-96.482,168.564,43.791,158.185
C06081=1030.839,69.418,-96.499,168.567,43.790,158.185
C06082=1030.846,69.667,-96.517,168.569,43.789,158.185
C06083=1030.852,69.917,-96.535,168.571,43.787,158.185
C06084=1030.858,70.166,-96.552,168.574,43.785,158.184
C06085=1030.864,70.415,-96.571,168.576,43.784,158.184
C06086=1030.871,70.665,-96.588,168.578,43.782,158.184
C06087=1030.877,70.914,-96.606,168.581,43.780,158.184
C06088=1030.883,71.163,-96.624,168.583,43.779,158.184
C06089=1030.889,71.413,-96.642,168.585,43.777,158.184
C06090=1030.895,71.662,-96.660,168.587,43.775,158.184
C06091=1030.901,71.911,-96.677,168.590,43.774,158.184
C06092=1030.908,72.160,-96.696,168.592,43.772,158.184
C06093=1030.914,72.410,-96.714,168.594,43.771,158.183
C06094=1030.920,72.659,-96.731,168.597,43.769,158.183
C06095=1030.926,72.908,-96.750,168.599,43.767,158.183
C06096=1030.932,73.158,-96.768,168.601,43.766,158.183
C06097=1030.939,73.407,-96.786,168.604,43.764,158.183
C06098=1030.945,73.656,-96.804,168.606,43.763,158.183
C06099=1030.951,73.905,-96.821,168.608,43.761,158.183
C06100=1030.957,74.155,-96.840,168.611,43.759,158.183
C06101=1030.963,74.404,-96.858,168.613,43.757,158.182
C06102=1030.969,74.653,-96.876,168.616,43.756,158.182
C06103=1030.976,74.902,-96.894,168.618,43.754,158.182
C06104=1030.982,75.152,-96.912,168.620,43.752,158.182
C06105=1030.989,75.401,-96.930,168.623,43.751,158.182
C06106=1030.994,75.650,-96.948,168.625,43.749,158.182
C06107=1031.001,75.935,-96.968,168.627,43.748,158.182
C06108=1031.009,76.221,-96.989,168.630,43.746,158.182
C06109=1031.016,76.506,-97.010,168.633,43.744,158.182
C06110=1031.023,76.792,-97.031,168.635,43.742,158.181
C06111=1031.029,77.041,-97.049,168.638,43.740,158.181
C06112=1031.035,77.290,-97.068,168.640,43.738,158.181
C06113=1031.042,77.540,-97.085,168.642,43.737,158.181
C06114=1031.048,77.789,-97.104,168.645,43.735,158.181
C06115=1031.054,78.038,-97.121,168.647,43.733,158.181
C06116=1031.060,78.288,-97.140,168.649,43.732,158.181
C06117=1031.066,78.537,-97.158,168.652,43.731,158.181
C06118=1031.072,78.786,-97.177,168.655,43.729,158.181
C06119=1031.078,79.036,-97.195,168.656,43.728,158.180
C06120=1031.084,79.285,-97.213,168.659,43.726,158.180
C06121=1031.091,79.534,-97.232,168.662,43.725,158.180
C06122=1031.097,79.783,-97.250,168.663,43.723,158.180
C06123=1031.103,80.033,-97.268,168.666,43.721,158.180
C06124=1031.109,80.282,-97.286,168.669,43.720,158.180
C06125=1031.115,80.531,-97.305,168.670,43.718,158.180
C06126=1031.121,80.780,-97.324,168.673,43.717,158.180
C06127=1031.127,81.030,-97.342,168.676,43.715,158.180
C06128=1031.133,81.279,-97.361,168.677,43.713,158.180
C06129=1031.140,81.528,-97.379,168.680,43.712,158.180
C06130=1031.145,81.777,-97.397,168.682,43.710,158.179
C06131=1031.152,82.026,-97.415,168.684,43.708,158.179
C06132=1031.158,82.275,-97.434,168.687,43.707,158.179
C06133=1031.164,82.525,-97.452,168.689,43.706,158.179
C06134=1031.170,82.775,-97.471,168.691,43.704,158.179
C06135=1031.176,83.024,-97.490,168.694,43.703,158.179
C06136=1031.182,83.273,-97.508,168.696,43.701,158.179
C06137=1031.188,83.522,-97.526,168.699,43.699,158.179
C06138=1031.195,83.771,-97.545,168.701,43.698,158.179
C06139=1031.201,84.020,-97.563,168.703,43.696,158.178
C06140=1031.207,84.270,-97.581,168.706,43.694,158.178
C06141=1031.214,84.519,-97.600,168.708,43.693,158.178
C06142=1031.219,84.768,-97.619,168.710,43.691,158.178
C06143=1031.226,85.018,-97.638,168.713,43.689,158.178
C06144=1031.232,85.267,-97.656,168.715,43.688,158.178
C06145=1031.238,85.516,-97.674,168.717,43.686,158.178
C06146=1031.244,85.765,-97.693,168.720,43.685,158.178
C06147=1031.251,86.014,-97.711,168.722,43.683,158.178
C06148=1031.257,86.264,-97.729,168.724,43.682,158.177
C06149=1031.263,86.513,-97.748,168.727,43.680,158.177
C06150=1031.269,86.762,-97.767,168.729,43.678,158.177
C06151=1031.275,87.011,-97.786,168.732,43.677,158.177
C06152=1031.282,87.260,-97.804,168.734,43.675,158.177
C06153=1031.288,87.510,-97.823,168.736,43.673,158.177
C06154=1031.294,87.759,-97.841,168.739,43.672,158.177
C06155=1031.301,88.008,-97.860,168.741,43.670,158.177
C06156=1031.307,88.258,-97.878,168.743,43.668,158.176
C06157=1031.313,88.507,-97.898,168.746,43.667,158.176
C06158=1031.319,88.756,-97.916,168.748,43.666,158.176
C06159=1031.325,89.005,-97.935,168.750,43.664,158.176
C06160=1031.331,89.254,-97.952,168.753,43.662,158.176
C06161=1031.337,89.503,-97.971,168.755,43.661,158.176
C06162=1031.344,89.753,-97.990,168.757,43.659,158.176
C06163=1031.350,90.002,-98.009,168.760,43.657,158.176
C06164=1031.356,90.251,-98.028,168.762,43.656,158.176
C06165=1031.362,90.501,-98.047,168.765,43.654,158.175
C06166=1031.368,90.750,-98.066,168.767,43.652,158.175
C06167=1031.374,90.999,-98.085,168.769,43.651,158.175
C06168=1031.380,91.248,-98.103,168.772,43.649,158.175
C06169=1031.387,91.497,-98.122,168.774,43.648,158.175
C06170=1031.392,91.747,-98.141,168.776,43.646,158.175
C06171=1031.399,92.032,-98.163,168.779,43.645,158.175
C06172=1031.406,92.318,-98.185,168.781,43.643,158.175
C06173=1031.414,92.603,-98.206,168.784,43.642,158.175
C06174=1031.421,92.888,-98.228,168.788,43.639,158.175
C06175=1031.426,93.137,-98.248,168.789,43.638,158.174
C06176=1031.433,93.386,-98.266,168.792,43.637,158.174
C06177=1031.439,93.636,-98.285,168.795,43.635,158.174
C06178=1031.445,93.885,-98.304,168.796,43.633,158.174
C06179=1031.451,94.134,-98.323,168.799,43.632,158.174
C06180=1031.457,94.383,-98.342,168.802,43.630,158.174
C06181=1031.464,94.633,-98.361,168.804,43.629,158.174
C06182=1031.469,94.882,-98.380,168.806,43.627,158.174
C06183=1031.476,95.131,-98.398,168.809,43.625,158.174
C06184=1031.482,95.380,-98.418,168.811,43.624,158.174
C06185=1031.488,95.629,-98.437,168.813,43.622,158.173
C06186=1031.494,95.878,-98.456,168.816,43.620,158.173
C06187=1031.500,96.128,-98.475,168.818,43.619,158.173
C06188=1031.507,96.377,-98.494,168.820,43.618,158.173
C06189=1031.512,96.626,-98.513,168.823,43.616,158.173
C06190=1031.519,96.875,-98.532,168.825,43.615,158.173
C06191=1031.525,97.124,-98.551,168.827,43.613,158.173
C06192=1031.532,97.374,-98.571,168.830,43.612,158.173
C06193=1031.537,97.623,-98.590,168.832,43.610,158.173
C06194=1031.544,97.872,-98.608,168.834,43.608,158.172
C06195=1031.550,98.122,-98.628,168.837,43.607,158.172
C06196=1031.556,98.370,-98.647,168.840,43.605,158.172
C06197=1031.562,98.620,-98.666,168.841,43.603,158.172
C06198=1031.568,98.869,-98.685,168.844,43.602,158.172
C06199=1031.574,99.118,-98.704,168.847,43.600,158.172
C06200=1031.581,99.367,-98.724,168.848,43.599,158.172
C06201=1031.587,99.616,-98.742,168.851,43.597,158.172
C06202=1031.593,99.865,-98.761,168.854,43.595,158.172
C06203=1031.599,100.116,-98.781,168.856,43.594,158.171
C06204=1031.606,100.364,-98.800,168.858,43.593,158.171
C06205=1031.612,100.613,-98.820,168.861,43.591,158.171
C06206=1031.617,100.863,-98.839,168.863,43.590,158.171
C06207=1031.623,101.112,-98.859,168.865,43.588,158.171
C06208=1031.630,101.361,-98.877,168.868,43.587,158.171
C06209=1031.635,101.610,-98.897,168.870,43.585,158.171
C06210=1031.641,101.859,-98.917,168.873,43.584,158.171
C06211=1031.647,102.109,-98.936,168.875,43.582,158.171
C06212=1031.654,102.357,-98.955,168.877,43.581,158.171
C06213=1031.660,102.607,-98.975,168.880,43.579,158.171
C06214=1031.666,102.856,-98.995,168.883,43.578,158.171
C06215=1031.673,103.105,-99.013,168.884,43.576,158.170
C06216=1031.678,103.355,-99.033,168.887,43.575,158.170
C06217=1031.684,103.603,-99.053,168.890,43.573,158.170
C06218=1031.690,103.853,-99.072,168.891,43.572,158.170
C06219=1031.697,104.101,-99.091,168.894,43.570,158.170
C06220=1031.702,104.351,-99.111,168.897,43.568,158.170
C06221=1031.709,104.600,-99.131,168.899,43.567,158.170
C06222=1031.715,104.850,-99.150,168.901,43.565,158.170
C06223=1031.721,105.098,-99.169,168.904,43.564,158.170
C06224=1031.727,105.348,-99.189,168.907,43.562,158.170
C06225=1031.733,105.596,-99.209,168.908,43.561,158.169
C06226=1031.739,105.846,-99.228,168.911,43.560,158.169
C06227=1031.746,106.095,-99.248,168.914,43.558,158.169
C06228=1031.752,106.344,-99.267,168.915,43.557,158.169
C06229=1031.758,106.593,-99.287,168.918,43.555,158.169
C06230=1031.763,106.843,-99.306,168.921,43.554,158.169
C06231=1031.770,107.091,-99.325,168.923,43.552,158.169
C06232=1031.776,107.341,-99.345,168.925,43.551,158.169
C06233=1031.782,107.590,-99.365,168.928,43.549,158.169
C06234=1031.788,107.840,-99.384,168.931,43.547,158.168
C06235=1031.795,108.124,-99.407,168.933,43.546,158.168
C06236=1031.803,108.410,-99.429,168.936,43.544,158.168
C06237=1031.810,108.695,-99.452,168.939,43.542,158.168
C06238=1031.816,108.981,-99.474,168.941,43.540,158.168
C06239=1031.823,109.229,-99.494,168.944,43.539,158.168
C06240=1031.829,109.479,-99.513,168.947,43.537,158.168
C06241=1031.835,109.728,-99.533,168.948,43.535,158.168
C06242=1031.841,109.977,-99.553,168.951,43.534,158.168
C06243=1031.847,110.226,-99.572,168.954,43.532,158.168
C06244=1031.854,110.476,-99.593,168.955,43.531,158.168
C06245=1031.860,110.724,-99.612,168.958,43.530,158.167
C06246=1031.866,110.974,-99.631,168.961,43.528,158.167
C06247=1031.872,111.223,-99.651,168.964,43.527,158.167
C06248=1031.879,111.472,-99.672,168.965,43.525,158.167
C06249=1031.884,111.722,-99.691,168.968,43.524,158.167
C06250=1031.890,111.970,-99.711,168.971,43.522,158.167
C06251=1031.896,112.219,-99.731,168.972,43.521,158.167
C06252=1031.903,112.469,-99.751,168.975,43.520,158.167
C06253=1031.909,112.718,-99.770,168.978,43.518,158.167
C06254=1031.914,112.967,-99.790,168.980,43.516,158.167
C06255=1031.921,113.216,-99.811,168.982,43.515,158.166
C06256=1031.927,113.465,-99.831,168.985,43.514,158.166
C06257=1031.933,113.714,-99.851,168.988,43.512,158.166
C06258=1031.938,113.964,-99.870,168.990,43.511,158.166
C06259=1031.945,114.213,-99.891,168.992,43.510,158.166
C06260=1031.951,114.462,-99.911,168.995,43.508,158.166
C06261=1031.957,114.711,-99.931,168.997,43.507,158.166
C06262=1031.963,114.960,-99.951,168.999,43.505,158.166
C06263=1031.968,115.210,-99.971,169.002,43.504,158.166
C06264=1031.974,115.458,-99.991,169.004,43.503,158.166
C06265=1031.980,115.707,-100.011,169.007,43.501,158.166
C06266=1031.986,115.956,-100.031,169.010,43.500,158.166
C06267=1031.992,116.206,-100.052,169.011,43.498,158.166
C06268=1031.998,116.455,-100.072,169.014,43.497,158.166
C06269=1032.004,116.704,-100.092,169.017,43.496,158.166
C06270=1032.011,116.953,-100.113,169.019,43.494,158.165
C06271=1032.017,117.202,-100.132,169.021,43.493,158.165
C06272=1032.022,117.452,-100.152,169.024,43.491,158.165
C06273=1032.028,117.700,-100.172,169.027,43.490,158.165
C06274=1032.034,117.950,-100.193,169.029,43.489,158.165
C06275=1032.040,118.199,-100.213,169.031,43.487,158.165
C06276=1032.046,118.448,-100.233,169.034,43.486,158.165
C06277=1032.052,118.697,-100.253,169.037,43.484,158.165
C06278=1032.058,118.946,-100.273,169.038,43.483,158.165
C06279=1032.065,119.194,-100.294,169.041,43.481,158.165
C06280=1032.071,119.444,-100.314,169.044,43.480,158.165
C06281=1032.076,119.693,-100.335,169.046,43.479,158.165
C06282=1032.082,119.942,-100.355,169.048,43.477,158.164
C06283=1032.089,120.191,-100.375,169.051,43.476,158.164
C06284=1032.095,120.440,-100.395,169.054,43.474,158.164
C06285=1032.101,120.690,-100.416,169.056,43.473,158.164
C06286=1032.107,120.939,-100.436,169.058,43.471,158.164
C06287=1032.113,121.188,-100.456,169.061,43.470,158.164
C06288=1032.119,121.437,-100.476,169.064,43.468,158.164
C06289=1032.125,121.686,-100.497,169.065,43.467,158.164
C06290=1032.131,121.935,-100.517,169.068,43.466,158.164
C06291=1032.137,122.185,-100.537,169.071,43.464,158.164
C06292=1032.144,122.433,-100.558,169.074,43.463,158.164
C06293=1032.149,122.683,-100.579,169.075,43.461,158.164
C06294=1032.155,122.931,-100.599,169.078,43.460,158.164
C06295=1032.162,123.181,-100.619,169.081,43.459,158.164
C06296=1032.168,123.430,-100.639,169.084,43.457,158.163
C06297=1032.173,123.679,-100.660,169.085,43.456,158.163
C06298=1032.180,123.928,-100.680,169.088,43.454,158.163
C06299=1032.187,124.214,-100.704,169.091,43.452,158.163
C06300=1032.194,124.498,-100.726,169.093,43.451,158.163
C06301=1032.201,124.784,-100.750,169.097,43.449,158.163
C06302=1032.208,125.069,-100.774,169.100,43.447,158.163
C06303=1032.214,125.318,-100.794,169.103,43.446,158.163
C06304=1032.221,125.567,-100.814,169.104,43.445,158.163
C06305=1032.226,125.816,-100.835,169.107,43.443,158.163
C06306=1032.233,126.065,-100.855,169.110,43.442,158.163
C06307=1032.239,126.314,-100.875,169.112,43.440,158.162
C06308=1032.245,126.564,-100.896,169.114,43.439,158.162
C06309=1032.251,126.812,-100.917,169.117,43.437,158.162
C06310=1032.258,127.062,-100.937,169.120,43.436,158.162
C06311=1032.264,127.310,-100.957,169.122,43.434,158.162
C06312=1032.269,127.560,-100.978,169.125,43.433,158.162
C06313=1032.276,127.808,-100.999,169.127,43.431,158.162
C06314=1032.282,128.058,-101.019,169.130,43.430,158.162
C06315=1032.288,128.307,-101.039,169.132,43.428,158.162
C06316=1032.294,128.556,-101.061,169.135,43.427,158.162
C06317=1032.300,128.805,-101.081,169.138,43.425,158.162
C06318=1032.307,129.054,-101.101,169.139,43.424,158.161
C06319=1032.313,129.303,-101.122,169.142,43.422,158.161
C06320=1032.319,129.552,-101.143,169.145,43.421,158.161
C06321=1032.326,129.802,-101.163,169.148,43.419,158.161
C06322=1032.332,130.050,-101.184,169.150,43.418,158.161
C06323=1032.338,130.300,-101.205,169.153,43.417,158.161
C06324=1032.344,130.549,-101.225,169.155,43.415,158.161
C06325=1032.351,130.798,-101.246,169.158,43.414,158.161
C06326=1032.356,131.047,-101.266,169.160,43.412,158.161
C06327=1032.362,131.296,-101.288,169.163,43.411,158.161
C06328=1032.368,131.545,-101.308,169.166,43.410,158.161
C06329=1032.374,131.794,-101.329,169.168,43.408,158.161
C06330=1032.380,132.043,-101.349,169.170,43.407,158.161
C06331=1032.387,132.292,-101.371,169.173,43.406,158.161
C06332=1032.392,132.541,-101.392,169.176,43.404,158.160
C06333=1032.399,132.790,-101.413,169.178,43.403,158.160
C06334=1032.405,133.040,-101.433,169.180,43.402,158.160
C06335=1032.411,133.288,-101.454,169.183,43.400,158.160
C06336=1032.417,133.538,-101.475,169.186,43.399,158.160
C06337=1032.422,133.786,-101.496,169.189,43.397,158.160
C06338=1032.429,134.035,-101.517,169.191,43.396,158.160
C06339=1032.434,134.284,-101.538,169.193,43.395,158.160
C06340=1032.441,134.533,-101.559,169.196,43.393,158.160
C06341=1032.447,134.783,-101.580,169.199,43.392,158.160
C06342=1032.453,135.032,-101.601,169.201,43.390,158.160
C06343=1032.460,135.280,-101.622,169.203,43.389,158.160
C06344=1032.465,135.530,-101.643,169.206,43.388,158.160
C06345=1032.471,135.779,-101.664,169.209,43.386,158.160
C06346=1032.478,136.028,-101.685,169.212,43.385,158.160
C06347=1032.483,136.277,-101.706,169.214,43.384,158.160
C06348=1032.490,136.526,-101.727,169.217,43.382,158.159
C06349=1032.495,136.775,-101.748,169.219,43.381,158.159
C06350=1032.502,137.024,-101.769,169.222,43.380,158.159
C06351=1032.508,137.273,-101.790,169.224,43.378,158.159
C06352=1032.514,137.522,-101.811,169.227,43.377,158.159
C06353=1032.520,137.771,-101.832,169.230,43.376,158.159
C06354=1032.526,138.020,-101.854,169.232,43.374,158.159
C06355=1032.532,138.269,-101.875,169.234,43.373,158.159
C06356=1032.538,138.518,-101.896,169.237,43.372,158.159
C06357=1032.544,138.768,-101.917,169.240,43.370,158.159
C06358=1032.551,139.016,-101.938,169.243,43.369,158.159
C06359=1032.557,139.265,-101.960,169.245,43.367,158.159
C06360=1032.562,139.514,-101.981,169.247,43.366,158.159
C06361=1032.568,139.763,-102.002,169.250,43.365,158.159
C06362=1032.574,140.013,-102.023,169.253,43.363,158.159
C06363=1032.582,140.297,-102.048,169.256,43.362,158.159
C06364=1032.588,140.582,-102.073,169.258,43.361,158.159
C06365=1032.595,140.868,-102.096,169.262,43.359,158.159
C06366=1032.602,141.153,-102.121,169.265,43.358,158.159
C06367=1032.608,141.401,-102.142,169.268,43.357,158.159
C06368=1032.614,141.650,-102.164,169.270,43.355,158.158
C06369=1032.621,141.900,-102.185,169.272,43.354,158.158
C06370=1032.626,142.148,-102.207,169.275,43.353,158.158
C06371=1032.632,142.398,-102.228,169.278,43.351,158.158
C06372=1032.638,142.647,-102.249,169.280,43.350,158.158
C06373=1032.644,142.896,-102.270,169.283,43.348,158.158
C06374=1032.650,143.145,-102.292,169.286,43.347,158.158
C06375=1032.657,143.394,-102.313,169.289,43.346,158.158
C06376=1032.663,143.643,-102.335,169.291,43.345,158.158
C06377=1032.668,143.891,-102.356,169.293,43.343,158.158
C06378=1032.675,144.141,-102.378,169.296,43.342,158.158
C06379=1032.681,144.390,-102.399,169.299,43.341,158.158
C06380=1032.687,144.639,-102.421,169.302,43.340,158.158
C06381=1032.692,144.887,-102.442,169.304,43.338,158.158
C06382=1032.699,145.137,-102.464,169.307,43.337,158.158
C06383=1032.705,145.386,-102.485,169.309,43.336,158.158
C06384=1032.712,145.635,-102.507,169.312,43.334,158.158
C06385=1032.717,145.883,-102.528,169.315,43.333,158.158
C06386=1032.723,146.133,-102.549,169.317,43.331,158.157
C06387=1032.730,146.382,-102.571,169.320,43.330,158.157
C06388=1032.736,146.631,-102.593,169.323,43.329,158.157
C06389=1032.741,146.879,-102.614,169.326,43.328,158.157
C06390=1032.747,147.129,-102.636,169.329,43.327,158.157
C06391=1032.754,147.378,-102.657,169.330,43.325,158.157
C06392=1032.760,147.627,-102.679,169.333,43.324,158.157
C06393=1032.766,147.876,-102.701,169.336,43.323,158.157
C06394=1032.772,148.124,-102.722,169.339,43.321,158.157
C06395=1032.778,148.373,-102.744,169.342,43.320,158.157
C06396=1032.783,148.623,-102.766,169.344,43.319,158.157
C06397=1032.790,148.872,-102.788,169.347,43.318,158.157
C06398=1032.796,149.121,-102.810,169.350,43.316,158.157
C06399=1032.802,149.369,-102.832,169.353,43.315,158.157
C06400=1032.808,149.618,-102.853,169.355,43.314,158.157
C06401=1032.814,149.868,-102.875,169.357,43.313,158.157
C06402=1032.820,150.117,-102.897,169.360,43.312,158.157
C06403=1032.827,150.365,-102.919,169.363,43.310,158.157
C06404=1032.831,150.614,-102.941,169.366,43.309,158.157
C06405=1032.838,150.863,-102.962,169.369,43.308,158.157
C06406=1032.844,151.113,-102.984,169.372,43.307,158.157
C06407=1032.850,151.361,-103.006,169.374,43.306,158.157
C06408=1032.856,151.610,-103.028,169.377,43.304,158.157
C06409=1032.863,151.860,-103.050,169.379,43.303,158.157
C06410=1032.867,152.108,-103.071,169.382,43.302,158.157
C06411=1032.874,152.357,-103.094,169.385,43.300,158.157
C06412=1032.880,152.606,-103.115,169.387,43.299,158.157
C06413=1032.886,152.855,-103.137,169.390,43.298,158.157
C06414=1032.893,153.104,-103.159,169.393,43.297,158.157
C06415=1032.899,153.353,-103.181,169.396,43.296,158.157
C06416=1032.905,153.602,-103.203,169.399,43.295,158.157
C06417=1032.911,153.851,-103.226,169.401,43.293,158.156
C06418=1032.916,154.100,-103.247,169.404,43.292,158.156
C06419=1032.923,154.348,-103.269,169.407,43.290,158.156
C06420=1032.929,154.598,-103.291,169.409,43.289,158.156
C06421=1032.934,154.847,-103.313,169.412,43.288,158.156
C06422=1032.941,155.096,-103.336,169.414,43.287,158.156
C06423=1032.947,155.345,-103.357,169.417,43.286,158.156
C06424=1032.953,155.594,-103.380,169.420,43.285,158.156
C06425=1032.959,155.843,-103.402,169.423,43.284,158.156
C06426=1032.965,156.092,-103.424,169.426,43.282,158.156
C06427=1032.972,156.377,-103.449,169.429,43.281,158.156
C06428=1032.979,156.661,-103.475,169.432,43.280,158.156
C06429=1032.985,156.946,-103.500,169.435,43.279,158.156
C06430=1032.992,157.231,-103.525,169.438,43.277,158.156
C06431=1032.999,157.479,-103.548,169.441,43.276,158.156
C06432=1033.005,157.728,-103.569,169.444,43.274,158.156
C06433=1033.011,157.977,-103.592,169.446,43.273,158.156
C06434=1033.017,158.227,-103.614,169.449,43.272,158.156
C06435=1033.023,158.475,-103.636,169.452,43.271,158.156
C06436=1033.029,158.725,-103.659,169.455,43.270,158.156
C06437=1033.035,158.973,-103.681,169.458,43.269,158.156
C06438=1033.041,159.222,-103.703,169.461,43.267,158.156
C06439=1033.047,159.471,-103.725,169.463,43.266,158.156
C06440=1033.053,159.720,-103.748,169.466,43.265,158.156
C06441=1033.059,159.969,-103.770,169.469,43.264,158.156
C06442=1033.065,160.218,-103.793,169.472,43.263,158.156
C06443=1033.071,160.467,-103.815,169.475,43.262,158.156
C06444=1033.076,160.715,-103.838,169.478,43.261,158.156
C06445=1033.082,160.965,-103.860,169.481,43.260,158.156
C06446=1033.088,161.213,-103.882,169.483,43.259,158.156
C06447=1033.094,161.462,-103.905,169.485,43.258,158.156
C06448=1033.100,161.711,-103.928,169.488,43.257,158.156
C06449=1033.105,161.960,-103.951,169.491,43.256,158.156
C06450=1033.111,162.209,-103.973,169.494,43.255,158.156
C06451=1033.117,162.458,-103.996,169.497,43.254,158.156
C06452=1033.123,162.707,-104.019,169.500,43.253,158.156
C06453=1033.129,162.956,-104.042,169.503,43.252,158.156
C06454=1033.135,163.204,-104.064,169.505,43.251,158.156
C06455=1033.141,163.453,-104.087,169.508,43.250,158.156
C06456=1033.146,163.703,-104.109,169.511,43.248,158.156
C06457=1033.152,163.952,-104.132,169.514,43.248,158.156
C06458=1033.158,164.200,-104.155,169.517,43.247,158.156
C06459=1033.164,164.449,-104.178,169.520,43.245,158.156
C06460=1033.170,164.698,-104.201,169.523,43.244,158.156
C06461=1033.176,164.947,-104.223,169.526,43.244,158.156
C06462=1033.181,165.196,-104.246,169.529,43.243,158.156
C06463=1033.188,165.444,-104.269,169.531,43.241,158.156
C06464=1033.194,165.693,-104.292,169.534,43.240,158.156
C06465=1033.199,165.942,-104.315,169.536,43.239,158.156
C06466=1033.205,166.191,-104.338,169.539,43.239,158.157
C06467=1033.212,166.440,-104.360,169.542,43.238,158.156
C06468=1033.217,166.689,-104.383,169.545,43.236,158.156
C06469=1033.223,166.937,-104.406,169.548,43.235,158.156
C06470=1033.229,167.187,-104.429,169.550,43.234,158.156
C06471=1033.236,167.436,-104.452,169.553,43.233,158.157
C06472=1033.242,167.685,-104.474,169.556,43.232,158.157
C06473=1033.247,167.933,-104.497,169.559,43.231,158.157
C06474=1033.253,168.182,-104.520,169.562,43.230,158.157
C06475=1033.259,168.431,-104.543,169.565,43.229,158.157
C06476=1033.265,168.680,-104.566,169.568,43.228,158.157
C06477=1033.271,168.929,-104.589,169.571,43.227,158.157
C06478=1033.277,169.178,-104.612,169.573,43.226,158.157
C06479=1033.283,169.427,-104.635,169.578,43.225,158.157
C06480=1033.289,169.676,-104.658,169.580,43.224,158.157
C06481=1033.295,169.925,-104.680,169.583,43.223,158.157
C06482=1033.301,170.174,-104.703,169.586,43.222,158.157
C06483=1033.307,170.423,-104.726,169.589,43.221,158.157
C06484=1033.312,170.671,-104.749,169.592,43.220,158.157
C06485=1033.318,170.920,-104.773,169.595,43.219,158.157
C06486=1033.325,171.169,-104.795,169.598,43.218,158.157
C06487=1033.331,171.418,-104.818,169.600,43.217,158.157
C06488=1033.337,171.667,-104.841,169.603,43.216,158.157
C06489=1033.343,171.916,-104.864,169.606,43.215,158.157
C06490=1033.348,172.165,-104.887,169.609,43.214,158.157
C06491=1033.356,172.448,-104.914,169.612,43.212,158.157
C06492=1033.363,172.733,-104.940,169.616,43.211,158.157
C06493=1033.370,173.017,-104.966,169.620,43.210,158.157
C06494=1033.377,173.302,-104.993,169.623,43.209,158.157
C06495=1033.382,173.550,-105.016,169.625,43.208,158.157
C06496=1033.389,173.799,-105.038,169.628,43.207,158.157
C06497=1033.395,174.049,-105.062,169.631,43.206,158.157
C06498=1033.401,174.297,-105.085,169.634,43.205,158.157
C06499=1033.407,174.546,-105.108,169.637,43.204,158.157
C06500=1033.413,174.795,-105.131,169.641,43.203,158.157
C06501=1033.420,175.044,-105.154,169.644,43.202,158.157
C06502=1033.426,175.292,-105.178,169.647,43.201,158.157
C06503=1033.432,175.541,-105.200,169.650,43.200,158.157
C06504=1033.438,175.791,-105.224,169.652,43.199,158.157
C06505=1033.444,176.039,-105.247,169.655,43.198,158.157
C06506=1033.450,176.288,-105.270,169.658,43.197,158.157
C06507=1033.456,176.536,-105.293,169.661,43.196,158.157
C06508=1033.463,176.785,-105.317,169.664,43.195,158.157
C06509=1033.469,177.034,-105.340,169.668,43.194,158.158
C06510=1033.474,177.283,-105.363,169.671,43.193,158.158
C06511=1033.481,177.532,-105.387,169.674,43.192,158.158
C06512=1033.487,177.781,-105.410,169.676,43.190,158.158
C06513=1033.493,178.029,-105.433,169.679,43.190,158.158
C06514=1033.500,178.279,-105.456,169.682,43.189,158.158
C06515=1033.505,178.528,-105.479,169.685,43.188,158.158
C06516=1033.512,178.776,-105.503,169.689,43.187,158.158
C06517=1033.518,179.025,-105.526,169.692,43.186,158.158
C06518=1033.524,179.274,-105.550,169.695,43.185,158.158
C06519=1033.530,179.523,-105.573,169.698,43.183,158.158
C06520=1033.537,179.771,-105.596,169.701,43.183,158.158
C06521=1033.543,180.020,-105.619,169.704,43.182,158.158
C06522=1033.549,180.269,-105.643,169.707,43.180,158.158
C06523=1033.555,180.518,-105.666,169.710,43.180,158.158
C06524=1033.561,180.766,-105.690,169.713,43.179,158.158
C06525=1033.567,181.016,-105.713,169.716,43.177,158.158
C06526=1033.573,181.264,-105.737,169.719,43.177,158.158
C06527=1033.581,181.514,-105.759,169.722,43.176,158.158
C06528=1033.587,181.762,-105.783,169.726,43.174,158.158
C06529=1033.593,182.011,-105.806,169.729,43.173,158.158
C06530=1033.599,182.260,-105.830,169.732,43.173,158.158
C06531=1033.608,182.616,-105.863,169.737,43.171,158.158
C06532=1033.617,182.971,-105.897,169.740,43.170,158.158
C06533=1033.626,183.328,-105.930,169.745,43.168,158.158
C06534=1033.634,183.684,-105.965,169.749,43.168,158.159
C06535=1033.640,183.932,-105.989,169.752,43.166,158.159
C06536=1033.645,184.180,-106.013,169.756,43.166,158.159
C06537=1033.652,184.429,-106.037,169.759,43.165,158.159
C06538=1033.657,184.679,-106.060,169.762,43.164,158.159
C06539=1033.664,184.928,-106.084,169.765,43.164,158.159
C06540=1033.669,185.176,-106.109,169.768,43.162,158.159
C06541=1033.675,185.424,-106.132,169.771,43.162,158.159
C06542=1033.682,185.673,-106.156,169.774,43.161,158.159
C06543=1033.687,185.922,-106.181,169.777,43.160,158.159
C06544=1033.694,186.171,-106.205,169.781,43.159,158.159
C06545=1033.699,186.420,-106.229,169.784,43.159,158.159
C06546=1033.705,186.668,-106.252,169.787,43.158,158.159
C06547=1033.711,186.918,-106.277,169.790,43.157,158.160
C06548=1033.717,187.166,-106.300,169.793,43.157,158.160
C06549=1033.722,187.415,-106.325,169.796,43.156,158.160
C06550=1033.728,187.664,-106.348,169.800,43.155,158.160
C06551=1033.733,187.876,-106.369,169.802,43.155,158.160
C06552=1033.739,188.089,-106.390,169.805,43.153,158.160
C06553=1033.744,188.302,-106.411,169.808,43.153,158.160
C06554=1033.749,188.515,-106.431,169.811,43.152,158.160
C06555=1033.755,188.728,-106.452,169.813,43.152,158.160
C06556=1033.760,188.941,-106.473,169.816,43.151,158.160
C06557=1033.764,189.153,-106.493,169.819,43.150,158.160
C06558=1033.770,189.366,-106.514,169.821,43.150,158.160
C06559=1033.776,189.615,-106.538,169.824,43.149,158.160
C06560=1033.782,189.863,-106.562,169.827,43.148,158.161
C06561=1033.788,190.113,-106.587,169.831,43.148,158.161
C06562=1033.794,190.361,-106.610,169.833,43.146,158.161
C06563=1033.800,190.610,-106.635,169.837,43.146,158.161
C06564=1033.806,190.858,-106.659,169.840,43.145,158.161
C06565=1033.812,191.108,-106.683,169.844,43.145,158.161
C06566=1033.818,191.356,-106.707,169.846,43.144,158.161
C06567=1033.824,191.605,-106.732,169.849,43.143,158.161
C06568=1033.830,191.854,-106.756,169.853,43.142,158.161
C06569=1033.836,192.102,-106.781,169.856,43.141,158.161
C06570=1033.843,192.351,-106.805,169.859,43.141,158.162
C06571=1033.848,192.600,-106.829,169.862,43.140,158.162
C06572=1033.855,192.849,-106.853,169.866,43.139,158.162
C06573=1033.860,193.097,-106.877,169.869,43.138,158.162
C06574=1033.866,193.346,-106.901,169.872,43.138,158.162
C06575=1033.873,193.595,-106.926,169.876,43.137,158.162
C06576=1033.879,193.843,-106.950,169.879,43.136,158.162
C06577=1033.885,194.093,-106.975,169.882,43.135,158.162
C06578=1033.891,194.342,-106.999,169.885,43.135,158.162
C06579=1033.897,194.590,-107.023,169.889,43.134,158.163
C06580=1033.903,194.838,-107.048,169.892,43.134,158.163
C06581=1033.909,195.088,-107.072,169.895,43.132,158.163
C06582=1033.915,195.336,-107.096,169.899,43.132,158.163
C06583=1033.922,195.585,-107.121,169.902,43.131,158.163
C06584=1033.928,195.834,-107.145,169.905,43.131,158.163
C06585=1033.934,196.082,-107.170,169.908,43.129,158.163
C06586=1033.940,196.331,-107.194,169.912,43.129,158.163
C06587=1033.946,196.580,-107.219,169.915,43.128,158.163
C06588=1033.952,196.828,-107.243,169.918,43.128,158.163
C06589=1033.958,197.077,-107.267,169.922,43.126,158.163
C06590=1033.965,197.326,-107.292,169.925,43.126,158.164
C06591=1033.971,197.574,-107.316,169.928,43.125,158.164
C06592=1033.978,197.823,-107.341,169.932,43.125,158.164
C06593=1033.983,198.072,-107.366,169.935,43.124,158.164
C06594=1033.990,198.321,-107.390,169.938,43.123,158.164
C06595=1033.996,198.569,-107.415,169.942,43.122,158.164
C06596=1034.002,198.818,-107.439,169.945,43.122,158.164
C06597=1034.009,199.067,-107.464,169.948,43.121,158.164
C06598=1034.014,199.316,-107.489,169.952,43.121,158.165
C06599=1034.021,199.564,-107.513,169.955,43.120,158.165
C06600=1034.027,199.813,-107.538,169.958,43.119,158.165
C06601=1034.034,200.061,-107.562,169.962,43.118,158.165
C06602=1034.040,200.311,-107.587,169.965,43.118,158.165
C06603=1034.046,200.560,-107.611,169.969,43.117,158.165
C06604=1034.052,200.808,-107.636,169.972,43.116,158.165
C06605=1034.058,201.056,-107.661,169.975,43.116,158.165
C06606=1034.064,201.305,-107.686,169.979,43.115,158.166
C06607=1034.070,201.554,-107.711,169.982,43.115,158.166
C06608=1034.077,201.802,-107.736,169.985,43.114,158.166
C06609=1034.082,202.051,-107.760,169.990,43.113,158.166
C06610=1034.089,202.300,-107.786,169.993,43.113,158.166
C06611=1034.095,202.548,-107.811,169.996,43.112,158.166
C06612=1034.101,202.798,-107.836,170.000,43.112,158.166
C06613=1034.107,203.046,-107.861,170.003,43.111,158.167
C06614=1034.112,203.294,-107.886,170.006,43.111,158.167
C06615=1034.118,203.544,-107.911,170.010,43.110,158.167
C06616=1034.125,203.792,-107.936,170.013,43.109,158.167
C06617=1034.131,204.041,-107.961,170.017,43.109,158.167
C06618=1034.138,204.289,-107.986,170.020,43.108,158.167
C06619=1034.163,205.339,-108.092,170.348,43.213,158.214
C06620=1034.172,205.681,-108.128,170.352,43.213,158.215
C06621=1034.182,206.022,-108.164,170.355,43.214,158.215
C06622=1034.191,206.362,-108.200,170.358,43.214,158.215
C06623=1034.200,206.704,-108.236,170.361,43.214,158.216
C06624=1034.207,206.952,-108.262,170.365,43.214,158.216
C06625=1034.214,207.200,-108.289,170.367,43.214,158.216
C06626=1034.221,207.449,-108.316,170.369,43.214,158.216
C06627=1034.227,207.697,-108.342,170.371,43.215,158.217
C06628=1034.234,207.946,-108.369,170.375,43.215,158.217
C06629=1034.241,208.195,-108.395,170.377,43.215,158.217
C06630=1034.247,208.443,-108.422,170.379,43.215,158.217
C06631=1034.254,208.692,-108.448,170.381,43.216,158.218
C06632=1034.261,208.940,-108.474,170.385,43.216,158.218
C06633=1034.268,209.189,-108.501,170.387,43.216,158.218
C06634=1034.274,209.438,-108.528,170.389,43.216,158.218
C06635=1034.281,209.685,-108.555,170.391,43.217,158.219
C06636=1034.288,209.934,-108.581,170.395,43.217,158.219
C06637=1034.295,210.183,-108.608,170.397,43.217,158.219
C06638=1034.301,210.431,-108.634,170.399,43.217,158.219
C06639=1034.308,210.680,-108.661,170.402,43.217,158.220
C06640=1034.315,210.928,-108.688,170.405,43.218,158.220
C06641=1034.321,211.176,-108.714,170.407,43.218,158.220
C06642=1034.328,211.425,-108.741,170.409,43.218,158.220
C06643=1034.335,211.674,-108.768,170.412,43.218,158.221
C06644=1034.341,211.922,-108.795,170.415,43.219,158.221
C06645=1034.348,212.171,-108.822,170.417,43.219,158.221
C06646=1034.354,212.420,-108.849,170.419,43.220,158.221
C06647=1034.361,212.667,-108.875,170.422,43.220,158.222
C06648=1034.368,212.916,-108.902,170.425,43.220,158.222
C06649=1034.375,213.165,-108.929,170.427,43.220,158.222
C06650=1034.381,213.413,-108.956,170.430,43.220,158.222
C06651=1034.388,213.661,-108.983,170.432,43.221,158.223
C06652=1034.394,213.911,-109.010,170.435,43.221,158.223
C06653=1034.401,214.158,-109.036,170.438,43.221,158.223
C06654=1034.407,214.407,-109.063,170.440,43.221,158.223
C06655=1034.415,214.656,-109.090,170.442,43.222,158.224
C06656=1034.421,214.904,-109.117,170.445,43.222,158.224
C06657=1034.428,215.152,-109.144,170.448,43.222,158.224
C06658=1034.434,215.401,-109.171,170.450,43.222,158.224
C06659=1034.442,215.649,-109.198,170.453,43.223,158.225
C06660=1034.448,215.898,-109.225,170.456,43.223,158.225
C06661=1034.455,216.146,-109.251,170.458,43.224,158.225
C06662=1034.461,216.395,-109.278,170.460,43.224,158.225
C06663=1034.469,216.643,-109.306,170.464,43.224,158.226
C06664=1034.475,216.892,-109.333,170.466,43.224,158.226
C06665=1034.482,217.140,-109.359,170.468,43.225,158.226
C06666=1034.488,217.389,-109.386,170.471,43.225,158.226
C06667=1034.496,217.637,-109.414,170.474,43.225,158.227
C06668=1034.502,217.886,-109.441,170.477,43.225,158.227
C06669=1034.509,218.134,-109.468,170.479,43.225,158.227
C06670=1034.515,218.382,-109.494,170.481,43.226,158.227
C06671=1034.523,218.631,-109.521,170.485,43.226,158.228
C06672=1034.529,218.880,-109.548,170.487,43.226,158.228
C06673=1034.536,219.128,-109.576,170.489,43.227,158.228
C06674=1034.543,219.376,-109.603,170.492,43.227,158.229
C06675=1034.549,219.625,-109.630,170.495,43.227,158.229
C06676=1034.559,219.971,-109.669,170.498,43.227,158.229
C06677=1034.568,220.318,-109.706,170.502,43.228,158.230
C06678=1034.577,220.666,-109.744,170.506,43.229,158.230
C06679=1034.586,221.012,-109.782,170.509,43.229,158.230
C06680=1034.593,221.260,-109.810,170.513,43.229,158.231
C06681=1034.599,221.510,-109.837,170.515,43.230,158.231
C06682=1034.606,221.757,-109.864,170.517,43.230,158.231
C06683=1034.613,222.005,-109.892,170.520,43.230,158.231
C06684=1034.620,222.254,-109.919,170.523,43.230,158.232
C06685=1034.626,222.503,-109.946,170.525,43.231,158.232
C06686=1034.633,222.751,-109.974,170.528,43.231,158.232
C06687=1034.640,222.999,-110.001,170.531,43.232,158.233
C06688=1034.646,223.247,-110.029,170.534,43.232,158.233
C06689=1034.653,223.496,-110.056,170.536,43.232,158.233
C06690=1034.659,223.745,-110.083,170.538,43.232,158.233
C06691=1034.666,223.993,-110.111,170.542,43.233,158.234
C06692=1034.673,224.242,-110.139,170.544,43.233,158.234
C06693=1034.680,224.490,-110.166,170.547,43.233,158.234
C06694=1034.687,224.738,-110.194,170.549,43.234,158.234
C06695=1034.693,224.987,-110.221,170.553,43.234,158.235
C06696=1034.700,225.236,-110.248,170.555,43.235,158.235
C06697=1034.706,225.484,-110.276,170.557,43.235,158.235
C06698=1034.713,225.732,-110.303,170.561,43.235,158.236
C06699=1034.720,225.980,-110.331,170.563,43.235,158.236
C06700=1034.727,226.228,-110.358,170.566,43.235,158.236
C06701=1034.733,226.477,-110.386,170.569,43.236,158.237
C06702=1034.740,226.725,-110.414,170.572,43.236,158.237
C06703=1034.746,226.974,-110.441,170.574,43.237,158.237
C06704=1034.754,227.223,-110.468,170.576,43.237,158.237
C06705=1034.760,227.471,-110.496,170.580,43.237,158.238
C06706=1034.767,227.719,-110.524,170.582,43.238,158.238
C06707=1034.774,227.968,-110.551,170.585,43.238,158.238
C06708=1034.781,228.216,-110.579,170.587,43.238,158.238
C06709=1034.787,228.465,-110.607,170.591,43.238,158.239
C06710=1034.794,228.713,-110.634,170.593,43.239,158.239
C06711=1034.801,228.962,-110.662,170.596,43.239,158.239
C06712=1034.807,229.210,-110.690,170.599,43.240,158.240
C06713=1034.814,229.458,-110.718,170.601,43.241,158.240
C06714=1034.821,229.706,-110.746,170.604,43.241,158.240
C06715=1034.828,229.955,-110.774,170.607,43.241,158.241
C06716=1034.834,230.203,-110.802,170.610,43.242,158.241
C06717=1034.841,230.452,-110.829,170.612,43.242,158.241
C06718=1034.847,230.700,-110.858,170.616,43.242,158.241
C06719=1034.854,230.949,-110.885,170.618,43.243,158.242
C06720=1034.860,231.197,-110.913,170.621,43.243,158.242
C06721=1034.867,231.445,-110.942,170.624,43.243,158.242
C06722=1034.874,231.694,-110.969,170.627,43.243,158.243
C06723=1034.881,231.942,-110.997,170.629,43.244,158.243
C06724=1034.887,232.190,-111.025,170.632,43.244,158.243
C06725=1034.894,232.439,-111.052,170.635,43.245,158.244
C06726=1034.900,232.687,-111.081,170.637,43.245,158.244
C06727=1034.907,232.935,-111.109,170.640,43.246,158.244
C06728=1034.914,233.184,-111.137,170.643,43.246,158.245
C06729=1034.921,233.432,-111.165,170.646,43.247,158.245
C06730=1034.927,233.680,-111.194,170.649,43.247,158.245
C06731=1034.933,233.929,-111.221,170.652,43.248,158.245
C06732=1034.942,234.268,-111.259,170.655,43.248,158.246
C06733=1034.952,234.607,-111.298,170.660,43.249,158.246
C06734=1034.960,234.947,-111.337,170.663,43.250,158.247
C06735=1034.970,235.286,-111.375,170.668,43.249,158.247
C06736=1034.976,235.534,-111.403,170.670,43.250,158.248
C06737=1034.983,235.783,-111.431,170.673,43.250,158.248
C06738=1034.990,236.030,-111.459,170.676,43.251,158.248
C06739=1034.996,236.279,-111.488,170.679,43.251,158.248
C06740=1035.003,236.528,-111.515,170.681,43.252,158.249
C06741=1035.010,236.775,-111.544,170.685,43.252,158.249
C06742=1035.017,237.025,-111.572,170.687,43.253,158.249
C06743=1035.023,237.273,-111.601,170.690,43.253,158.250
C06744=1035.030,237.521,-111.629,170.693,43.254,158.250
C06745=1035.037,237.769,-111.657,170.696,43.254,158.250
C06746=1035.044,238.017,-111.685,170.698,43.255,158.251
C06747=1035.050,238.265,-111.714,170.702,43.255,158.251
C06748=1035.056,238.514,-111.742,170.705,43.255,158.251
C06749=1035.064,238.762,-111.770,170.707,43.256,158.252
C06750=1035.070,239.011,-111.799,170.711,43.256,158.252
C06751=1035.077,239.259,-111.827,170.713,43.257,158.252
C06752=1035.084,239.507,-111.855,170.716,43.257,158.253
C06753=1035.090,239.756,-111.884,170.719,43.258,158.253
C06754=1035.097,240.004,-111.912,170.722,43.258,158.253
C06755=1035.104,240.252,-111.940,170.724,43.259,158.254
C06756=1035.111,240.500,-111.969,170.728,43.259,158.254
C06757=1035.117,240.749,-111.997,170.731,43.259,158.254
C06758=1035.124,240.997,-112.026,170.733,43.260,158.255
C06759=1035.130,241.245,-112.055,170.737,43.260,158.255
C06760=1035.136,241.494,-112.083,170.739,43.261,158.255
C06761=1035.143,241.742,-112.112,170.742,43.261,158.256
C06762=1035.150,241.990,-112.141,170.745,43.262,158.256
C06763=1035.157,242.239,-112.169,170.748,43.262,158.256
C06764=1035.163,242.487,-112.198,170.751,43.263,158.257
C06765=1035.170,242.735,-112.226,170.754,43.263,158.257
C06766=1035.176,242.983,-112.255,170.757,43.264,158.257
C06767=1035.184,243.232,-112.283,170.760,43.264,158.258
C06768=1035.190,243.480,-112.312,170.763,43.265,158.258
C06769=1035.197,243.728,-112.341,170.765,43.265,158.258
C06770=1035.203,243.976,-112.370,170.769,43.266,158.259
C06771=1035.209,244.224,-112.399,170.772,43.266,158.259
C06772=1035.217,244.474,-112.427,170.774,43.267,158.259
C06773=1035.223,244.722,-112.456,170.778,43.268,158.260
C06774=1035.230,244.969,-112.484,170.780,43.268,158.260
C06775=1035.236,245.218,-112.513,170.784,43.269,158.260
C06776=1035.243,245.466,-112.543,170.787,43.269,158.261
C06777=1035.249,245.715,-112.572,170.789,43.270,158.261
C06778=1035.255,245.963,-112.601,170.793,43.270,158.261
C06779=1035.262,246.211,-112.630,170.795,43.271,158.262
C06780=1035.269,246.459,-112.658,170.799,43.271,158.262
C06781=1035.276,246.707,-112.688,170.802,43.272,158.263
C06782=1035.282,246.956,-112.717,170.804,43.273,158.263
C06783=1035.288,247.204,-112.746,170.808,43.273,158.263
C06784=1035.294,247.452,-112.775,170.810,43.274,158.264
C06785=1035.302,247.700,-112.804,170.814,43.275,158.264
C06786=1035.308,247.949,-112.833,170.817,43.275,158.264
C06787=1035.314,248.197,-112.862,170.819,43.276,158.265
C06788=1035.323,248.530,-112.901,170.824,43.277,158.265
C06789=1035.332,248.864,-112.940,170.827,43.278,158.266
C06790=1035.341,249.197,-112.980,170.832,43.278,158.266
C06791=1035.350,249.530,-113.018,170.835,43.279,158.267
C06792=1035.356,249.779,-113.047,170.839,43.280,158.267
C06793=1035.363,250.027,-113.077,170.842,43.280,158.268
C06794=1035.369,250.276,-113.106,170.845,43.281,158.268
C06795=1035.376,250.523,-113.136,170.848,43.281,158.268
C06796=1035.383,250.772,-113.164,170.852,43.282,158.269
C06797=1035.390,251.020,-113.194,170.854,43.283,158.269
C06798=1035.396,251.268,-113.223,170.857,43.283,158.269
C06799=1035.403,251.517,-113.252,170.861,43.284,158.270
C06800=1035.409,251.764,-113.282,170.863,43.284,158.270
C06801=1035.416,252.013,-113.311,170.867,43.285,158.270
C06802=1035.423,252.261,-113.340,170.870,43.285,158.271
C06803=1035.429,252.509,-113.369,170.872,43.286,158.271
C06804=1035.437,252.757,-113.399,170.876,43.287,158.272
C06805=1035.443,253.005,-113.428,170.879,43.288,158.272
C06806=1035.450,253.254,-113.457,170.882,43.288,158.272
C06807=1035.456,253.502,-113.486,170.885,43.289,158.273
C06808=1035.462,253.750,-113.516,170.888,43.289,158.273
C06809=1035.470,253.998,-113.545,170.892,43.290,158.274
C06810=1035.476,254.246,-113.574,170.894,43.290,158.274
C06811=1035.483,254.495,-113.604,170.898,43.291,158.274
C06812=1035.490,254.743,-113.633,170.901,43.292,158.275
C06813=1035.497,254.992,-113.662,170.904,43.293,158.275
C06814=1035.503,255.239,-113.692,170.907,43.293,158.275
C06815=1035.510,255.488,-113.722,170.910,43.293,158.276
C06816=1035.517,255.735,-113.751,170.914,43.294,158.276
C06817=1035.523,255.983,-113.780,170.916,43.295,158.277
C06818=1035.530,256.232,-113.809,170.919,43.295,158.277
C06819=1035.537,256.480,-113.839,170.923,43.296,158.277
C06820=1035.544,256.728,-113.868,170.926,43.296,158.278
C06821=1035.550,256.976,-113.898,170.929,43.297,158.278
C06822=1035.557,257.225,-113.927,170.932,43.298,158.278
C06823=1035.564,257.473,-113.958,170.936,43.298,158.279
C06824=1035.571,257.721,-113.986,170.939,43.299,158.279
C06825=1035.578,257.969,-114.016,170.942,43.299,158.280
C06826=1035.585,258.217,-114.045,170.945,43.300,158.280
C06827=1035.592,258.465,-114.075,170.948,43.300,158.280
C06828=1035.598,258.714,-114.104,170.952,43.301,158.281
C06829=1035.605,258.962,-114.135,170.955,43.302,158.281
C06830=1035.611,259.210,-114.164,170.958,43.303,158.281
C06831=1035.619,259.458,-114.194,170.961,43.303,158.282
C06832=1035.625,259.707,-114.223,170.964,43.303,158.282
C06833=1035.633,259.954,-114.252,170.968,43.304,158.283
C06834=1035.640,260.203,-114.282,170.971,43.305,158.283
C06835=1035.646,260.450,-114.311,170.974,43.306,158.283
C06836=1035.653,260.699,-114.342,170.977,43.306,158.284
C06837=1035.660,260.948,-114.371,170.981,43.307,158.284
C06838=1035.667,261.195,-114.401,170.984,43.307,158.285
C06839=1035.674,261.443,-114.431,170.987,43.308,158.285
C06840=1035.680,261.691,-114.460,170.991,43.309,158.285
C06841=1035.687,261.940,-114.490,170.993,43.310,158.286
C06842=1035.694,262.188,-114.520,170.997,43.310,158.286
C06843=1035.700,262.436,-114.550,171.000,43.311,158.287
C06844=1035.710,262.768,-114.591,171.005,43.312,158.287
C06845=1035.718,263.100,-114.630,171.008,43.313,158.288
C06846=1035.727,263.432,-114.670,171.013,43.314,158.288
C06847=1035.736,263.764,-114.711,171.018,43.315,158.289
C06848=1035.742,264.012,-114.741,171.021,43.316,158.289
C06849=1035.749,264.260,-114.771,171.025,43.316,158.290
C06850=1035.757,264.508,-114.801,171.027,43.317,158.290
C06851=1035.763,264.756,-114.831,171.031,43.318,158.291
C06852=1035.770,265.004,-114.862,171.034,43.319,158.291
C06853=1035.777,265.253,-114.892,171.038,43.319,158.291
C06854=1035.783,265.500,-114.922,171.041,43.320,158.292
C06855=1035.790,265.749,-114.952,171.045,43.321,158.292
C06856=1035.797,265.997,-114.982,171.047,43.322,158.293
C06857=1035.803,266.244,-115.012,171.050,43.322,158.293
C06858=1035.811,266.493,-115.042,171.054,43.323,158.294
C06859=1035.817,266.741,-115.073,171.057,43.324,158.294
C06860=1035.824,266.989,-115.103,171.061,43.324,158.294
C06861=1035.831,267.237,-115.133,171.064,43.325,158.295
C06862=1035.837,267.485,-115.164,171.068,43.327,158.295
C06863=1035.844,267.733,-115.193,171.070,43.327,158.296
C06864=1035.850,267.981,-115.224,171.074,43.328,158.296
C06865=1035.857,268.230,-115.254,171.077,43.329,158.297
C06866=1035.864,268.478,-115.286,171.081,43.329,158.297
C06867=1035.871,268.725,-115.315,171.084,43.330,158.298
C06868=1035.878,268.973,-115.345,171.088,43.331,158.298
C06869=1035.884,269.222,-115.376,171.092,43.332,158.299
C06870=1035.891,269.470,-115.406,171.095,43.333,158.299
C06871=1035.897,269.718,-115.437,171.097,43.334,158.299
C06872=1035.905,269.965,-115.467,171.101,43.334,158.300
C06873=1035.911,270.214,-115.498,171.104,43.335,158.300
C06874=1035.918,270.462,-115.528,171.108,43.336,158.301
C06875=1035.924,270.710,-115.559,171.112,43.337,158.301
C06876=1035.931,270.958,-115.589,171.115,43.338,158.302
C06877=1035.938,271.206,-115.620,171.118,43.339,158.302
C06878=1035.945,271.454,-115.650,171.122,43.339,158.303
C06879=1035.951,271.702,-115.681,171.125,43.340,158.303
C06880=1035.958,271.950,-115.712,171.128,43.341,158.304
C06881=1035.965,272.198,-115.742,171.132,43.342,158.304
C06882=1035.971,272.446,-115.774,171.135,43.343,158.304
C06883=1035.979,272.694,-115.804,171.139,43.343,158.305
C06884=1035.985,272.942,-115.835,171.142,43.345,158.305
C06885=1035.991,273.190,-115.866,171.146,43.345,158.306
C06886=1035.999,273.438,-115.896,171.149,43.346,158.306
C06887=1036.005,273.686,-115.927,171.153,43.347,158.307
C06888=1036.012,273.934,-115.958,171.156,43.348,158.307
C06889=1036.019,274.182,-115.989,171.160,43.349,158.308
C06890=1036.025,274.430,-116.020,171.163,43.350,158.308
C06891=1036.032,274.678,-116.050,171.167,43.351,158.309
C06892=1036.039,274.926,-116.081,171.170,43.352,158.309
C06893=1036.045,275.174,-116.112,171.174,43.352,158.310
C06894=1036.052,275.422,-116.143,171.177,43.354,158.310
C06895=1036.059,275.670,-116.174,171.180,43.354,158.311
C06896=1036.066,275.918,-116.205,171.184,43.356,158.311
C06897=1036.072,276.166,-116.235,171.187,43.356,158.312
C06898=1036.079,276.414,-116.266,171.191,43.357,158.312
C06899=1036.086,276.662,-116.298,171.194,43.358,158.313
C06900=1036.095,276.999,-116.340,171.199,43.360,158.313
C06901=1036.104,277.335,-116.381,171.204,43.361,158.314
C06902=1036.113,277.672,-116.424,171.208,43.362,158.314
C06903=1036.123,278.009,-116.466,171.214,43.363,158.315
C06904=1036.130,278.257,-116.497,171.218,43.364,158.316
C06905=1036.136,278.504,-116.528,171.220,43.365,158.316
C06906=1036.143,278.752,-116.560,171.224,43.366,158.317
C06907=1036.149,279.000,-116.591,171.227,43.367,158.317
C06908=1036.156,279.249,-116.622,171.231,43.368,158.318
C06909=1036.162,279.496,-116.653,171.235,43.369,158.318
C06910=1036.169,279.744,-116.685,171.238,43.370,158.319
C06911=1036.176,279.992,-116.716,171.242,43.371,158.319
C06912=1036.183,280.240,-116.747,171.245,43.372,158.320
C06913=1036.190,280.488,-116.778,171.249,43.373,158.320
C06914=1036.197,280.736,-116.810,171.253,43.374,158.321
C06915=1036.204,280.984,-116.841,171.256,43.375,158.321
C06916=1036.210,281.231,-116.873,171.260,43.376,158.322
C06917=1036.217,281.479,-116.904,171.263,43.377,158.322
C06918=1036.223,281.728,-116.935,171.267,43.378,158.323
C06919=1036.230,281.976,-116.966,171.272,43.379,158.323
C06920=1036.237,282.224,-116.998,171.275,43.380,158.324
C06921=1036.244,282.472,-117.029,171.279,43.381,158.324
C06922=1036.250,282.720,-117.060,171.282,43.382,158.325
C06923=1036.257,282.967,-117.092,171.286,43.383,158.325
C06924=1036.264,283.215,-117.124,171.290,43.385,158.326
C06925=1036.271,283.463,-117.155,171.293,43.385,158.326
C06926=1036.278,283.710,-117.187,171.297,43.386,158.327
C06927=1036.284,283.958,-117.218,171.300,43.387,158.327
C06928=1036.291,284.206,-117.250,171.304,43.388,158.328
C06929=1036.298,284.454,-117.281,171.308,43.390,158.329
C06930=1036.305,284.703,-117.313,171.311,43.390,158.329
C06931=1036.312,284.951,-117.344,171.315,43.392,158.330
C06932=1036.318,285.199,-117.376,171.318,43.392,158.330
C06933=1036.325,285.446,-117.408,171.322,43.394,158.331
C06934=1036.332,285.694,-117.439,171.326,43.395,158.331
C06935=1036.339,285.942,-117.471,171.330,43.396,158.332
C06936=1036.346,286.190,-117.502,171.334,43.397,158.332
C06937=1036.352,286.438,-117.534,171.338,43.398,158.333
C06938=1036.360,286.686,-117.566,171.341,43.399,158.333
C06939=1036.367,286.933,-117.598,171.345,43.400,158.334
C06940=1036.373,287.181,-117.629,171.348,43.401,158.334
C06941=1036.381,287.429,-117.661,171.352,43.402,158.335
C06942=1036.386,287.677,-117.693,171.356,43.403,158.335
C06943=1036.393,287.925,-117.725,171.359,43.405,158.336
C06944=1036.400,288.172,-117.757,171.364,43.406,158.337
C06945=1036.408,288.421,-117.789,171.367,43.406,158.337
C06946=1036.414,288.668,-117.820,171.371,43.408,158.338
C06947=1036.421,288.916,-117.853,171.375,43.409,158.338
C06948=1036.427,289.164,-117.884,171.379,43.410,158.339
C06949=1036.434,289.411,-117.916,171.382,43.412,158.339
C06950=1036.442,289.660,-117.948,171.386,43.412,158.340
C06951=1036.448,289.907,-117.981,171.389,43.414,158.340
C06952=1036.455,290.155,-118.012,171.394,43.415,158.341
C06953=1036.462,290.403,-118.045,171.398,43.416,158.342
C06954=1036.468,290.651,-118.076,171.402,43.417,158.342
C06955=1036.475,290.899,-118.109,171.405,43.419,158.343
C06956=1036.484,291.248,-118.154,171.410,43.420,158.344
C06957=1036.495,291.596,-118.199,171.416,43.422,158.344
C06958=1036.504,291.945,-118.244,171.421,43.424,158.345
C06959=1036.514,292.293,-118.290,171.427,43.425,158.346
C06960=1036.521,292.541,-118.322,171.431,43.426,158.347
C06961=1036.527,292.789,-118.354,171.434,43.428,158.347
C06962=1036.535,293.037,-118.386,171.438,43.429,158.348
C06963=1036.542,293.284,-118.418,171.443,43.430,158.348
C06964=1036.548,293.532,-118.450,171.446,43.431,158.349
C06965=1036.555,293.780,-118.483,171.450,43.433,158.350
C06966=1036.562,294.028,-118.516,171.454,43.433,158.350
C06967=1036.569,294.275,-118.548,171.457,43.435,158.351
C06968=1036.575,294.523,-118.580,171.462,43.436,158.351
C06969=1036.582,294.771,-118.612,171.466,43.437,158.352
C06970=1036.589,295.019,-118.645,171.469,43.438,158.352
C06971=1036.596,295.266,-118.677,171.473,43.440,158.353
C06972=1036.603,295.515,-118.710,171.477,43.441,158.354
C06973=1036.609,295.762,-118.743,171.481,43.443,158.354
C06974=1036.616,296.009,-118.775,171.485,43.444,158.355
C06975=1036.622,296.257,-118.808,171.489,43.445,158.356
C06976=1036.629,296.505,-118.841,171.493,43.446,158.356
C06977=1036.636,296.753,-118.873,171.497,43.448,158.357
C06978=1036.642,297.000,-118.906,171.500,43.450,158.357
C06979=1036.649,297.249,-118.939,171.505,43.451,158.358
C06980=1036.656,297.496,-118.972,171.509,43.452,158.359
C06981=1036.663,297.743,-119.004,171.513,43.453,158.359
C06982=1036.670,297.992,-119.037,171.516,43.455,158.360
C06983=1036.676,298.239,-119.070,171.521,43.456,158.361
C06984=1036.683,298.488,-119.103,171.525,43.457,158.361
C06985=1036.690,298.734,-119.136,171.529,43.459,158.362
C06986=1036.696,298.982,-119.169,171.532,43.460,158.362
C06987=1036.703,299.230,-119.202,171.536,43.462,158.363
C06988=1036.710,299.478,-119.234,171.541,43.463,158.364
C06989=1036.717,299.726,-119.267,171.545,43.464,158.364
C06990=1036.723,299.973,-119.300,171.548,43.466,158.365
C06991=1036.731,300.221,-119.334,171.553,43.467,158.366
C06992=1036.737,300.469,-119.366,171.557,43.469,158.366
C06993=1036.744,300.716,-119.398,171.561,43.470,158.367
C06994=1036.751,300.964,-119.432,171.565,43.472,158.368
C06995=1036.757,301.211,-119.465,171.569,43.473,158.368
C06996=1036.764,301.459,-119.498,171.573,43.474,158.369
C06997=1036.771,301.707,-119.531,171.577,43.475,158.369
C06998=1036.779,301.954,-119.564,171.582,43.477,158.370
C06999=1036.785,302.202,-119.597,171.585,43.478,158.371
C07000=1036.792,302.450,-119.630,171.589,43.480,158.371
C07001=1036.798,302.697,-119.663,171.593,43.481,158.372
C07002=1036.806,302.945,-119.696,171.598,43.483,158.373
C07003=1036.813,303.193,-119.730,171.602,43.484,158.374
C07004=1036.820,303.440,-119.762,171.605,43.486,158.374
C07005=1036.826,303.689,-119.796,171.610,43.487,158.375
C07006=1036.833,303.936,-119.829,171.614,43.489,158.376
C07007=1036.841,304.184,-119.862,171.618,43.490,158.376
C07008=1036.847,304.431,-119.895,171.622,43.491,158.377
C07009=1036.854,304.679,-119.928,171.626,43.493,158.378
C07010=1036.861,304.927,-119.962,171.630,43.494,158.378
C07011=1036.868,305.174,-119.995,171.635,43.496,158.379
C07012=1036.879,305.539,-120.043,171.641,43.498,158.380
C07013=1036.889,305.905,-120.092,171.647,43.500,158.381
C07014=1036.899,306.270,-120.142,171.653,43.502,158.382
C07015=1036.909,306.636,-120.191,171.660,43.504,158.383
C07016=1036.917,306.883,-120.224,171.663,43.506,158.383
C07017=1036.924,307.131,-120.258,171.668,43.507,158.384
C07018=1036.930,307.379,-120.291,171.672,43.509,158.385
C07019=1036.937,307.626,-120.325,171.676,43.510,158.386
C07020=1036.945,307.874,-120.358,171.680,43.512,158.386
C07021=1036.952,308.122,-120.391,171.684,43.513,158.387
C07022=1036.959,308.369,-120.425,171.689,43.514,158.388
C07023=1036.966,308.617,-120.458,171.693,43.516,158.388
C07024=1036.973,308.864,-120.492,171.698,43.517,158.389
C07025=1036.981,309.112,-120.525,171.702,43.519,158.390
C07026=1036.987,309.359,-120.558,171.706,43.521,158.390
C07027=1036.995,309.607,-120.592,171.710,43.522,158.391
C07028=1037.002,309.855,-120.626,171.714,43.524,158.392
C07029=1037.009,310.102,-120.660,171.719,43.525,158.392
C07030=1037.016,310.350,-120.693,171.723,43.527,158.393
C07031=1037.024,310.598,-120.726,171.728,43.528,158.394
C07032=1037.030,310.845,-120.759,171.732,43.530,158.395
C07033=1037.038,311.092,-120.793,171.736,43.532,158.395
C07034=1037.045,311.340,-120.827,171.740,43.533,158.396
C07035=1037.052,311.588,-120.861,171.745,43.535,158.397
C07036=1037.059,311.836,-120.895,171.749,43.536,158.397
C07037=1037.066,312.083,-120.929,171.754,43.538,158.398
C07038=1037.072,312.330,-120.963,171.758,43.539,158.399
C07039=1037.080,312.578,-120.996,171.763,43.541,158.400
C07040=1037.087,312.826,-121.030,171.767,43.543,158.400
C07041=1037.093,313.073,-121.065,171.770,43.545,158.401
C07042=1037.100,313.320,-121.099,171.775,43.547,158.402
C07043=1037.107,313.568,-121.133,171.779,43.548,158.403
C07044=1037.114,313.816,-121.167,171.784,43.550,158.403
C07045=1037.121,314.063,-121.202,171.788,43.552,158.404
C07046=1037.128,314.311,-121.236,171.793,43.554,158.405
C07047=1037.135,314.559,-121.270,171.797,43.555,158.406
C07048=1037.141,314.806,-121.304,171.802,43.557,158.406
C07049=1037.148,315.053,-121.338,171.806,43.558,158.407
C07050=1037.155,315.301,-121.373,171.811,43.560,158.408
C07051=1037.162,315.549,-121.407,171.815,43.562,158.409
C07052=1037.169,315.796,-121.441,171.820,43.564,158.410
C07053=1037.176,316.044,-121.476,171.824,43.566,158.410
C07054=1037.183,316.291,-121.510,171.828,43.567,158.411
C07055=1037.190,316.539,-121.545,171.832,43.569,158.412
C07056=1037.197,316.786,-121.578,171.837,43.571,158.413
C07057=1037.204,317.034,-121.614,171.841,43.573,158.414
C07058=1037.211,317.281,-121.647,171.846,43.575,158.414
C07059=1037.218,317.529,-121.683,171.850,43.577,158.415
C07060=1037.225,317.776,-121.716,171.855,43.578,158.416
C07061=1037.232,318.024,-121.752,171.859,43.580,158.417
C07062=1037.239,318.271,-121.785,171.864,43.582,158.417
C07063=1037.246,318.518,-121.820,171.868,43.584,158.418
C07064=1037.253,318.766,-121.854,171.873,43.585,158.419
C07065=1037.260,319.013,-121.889,171.878,43.587,158.420
C07066=1037.267,319.261,-121.924,171.882,43.589,158.420
C07067=1037.274,319.509,-121.958,171.887,43.591,158.421
C07068=1037.285,319.879,-122.010,171.894,43.594,158.423
C07069=1037.296,320.249,-122.062,171.900,43.597,158.424
C07070=1037.306,320.619,-122.113,171.907,43.599,158.425
C07071=1037.316,320.989,-122.165,171.914,43.602,158.426
C07072=1037.324,321.237,-122.200,171.919,43.604,158.427
C07073=1037.331,321.484,-122.235,171.923,43.606,158.428
C07074=1037.338,321.732,-122.269,171.928,43.608,158.429
C07075=1037.345,321.979,-122.304,171.933,43.609,158.429
C07076=1037.353,322.227,-122.339,171.937,43.612,158.430
C07077=1037.359,322.474,-122.374,171.942,43.613,158.431
C07078=1037.367,322.722,-122.409,171.947,43.615,158.432
C07079=1037.374,322.970,-122.443,171.951,43.617,158.433
C07080=1037.381,323.217,-122.478,171.956,43.619,158.434
C07081=1037.388,323.464,-122.513,171.961,43.621,158.434
C07082=1037.396,323.712,-122.548,171.965,43.623,158.435
C07083=1037.403,323.959,-122.583,171.970,43.625,158.436
C07084=1037.411,324.206,-122.617,171.975,43.627,158.437
C07085=1037.417,324.454,-122.653,171.979,43.628,158.438
C07086=1037.425,324.701,-122.687,171.984,43.631,158.439
C07087=1037.432,324.949,-122.723,171.989,43.632,158.439
C07088=1037.440,325.196,-122.757,171.993,43.634,158.440
C07089=1037.447,325.444,-122.793,171.998,43.636,158.441
C07090=1037.455,325.691,-122.827,172.003,43.638,158.442
C07091=1037.461,325.938,-122.862,172.008,43.640,158.443
C07092=1037.469,326.186,-122.897,172.012,43.642,158.444
C07093=1037.476,326.433,-122.932,172.017,43.644,158.444
C07094=1037.484,326.680,-122.967,172.022,43.646,158.445
C07095=1037.491,326.928,-123.002,172.027,43.648,158.446
C07096=1037.498,327.176,-123.038,172.031,43.650,158.447
C07097=1037.506,327.424,-123.072,172.036,43.652,158.448
C07098=1037.513,327.670,-123.108,172.042,43.654,158.449
C07099=1037.521,327.917,-123.143,172.046,43.656,158.450
C07100=1037.528,328.165,-123.178,172.051,43.658,158.451
C07101=1037.535,328.413,-123.213,172.056,43.660,158.451
C07102=1037.543,328.661,-123.248,172.061,43.662,158.452
C07103=1037.550,328.907,-123.284,172.066,43.664,158.453
C07104=1037.557,329.155,-123.320,172.070,43.666,158.454
C07105=1037.564,329.402,-123.356,172.075,43.668,158.455
C07106=1037.571,329.649,-123.391,172.080,43.671,158.456
C07107=1037.578,329.898,-123.426,172.085,43.672,158.457
C07108=1037.586,330.144,-123.462,172.089,43.675,158.458
C07109=1037.593,330.392,-123.498,172.095,43.677,158.459
C07110=1037.600,330.639,-123.533,172.100,43.679,158.460
C07111=1037.607,330.887,-123.569,172.105,43.681,158.460
C07112=1037.615,331.134,-123.604,172.109,43.683,158.461
C07113=1037.623,331.381,-123.640,172.114,43.686,158.462
C07114=1037.630,331.628,-123.675,172.119,43.688,158.463
C07115=1037.637,331.876,-123.712,172.124,43.690,158.464
C07116=1037.644,332.123,-123.747,172.130,43.692,158.465
C07117=1037.652,332.371,-123.783,172.134,43.694,158.466
C07118=1037.659,332.617,-123.819,172.139,43.696,158.467
C07119=1037.666,332.865,-123.854,172.144,43.699,158.468
C07120=1037.673,333.112,-123.890,172.149,43.701,158.469
C07121=1037.681,333.360,-123.926,172.154,43.703,158.470
C07122=1037.688,333.607,-123.962,172.159,43.705,158.471
C07123=1037.695,333.854,-123.998,172.164,43.708,158.472
C07124=1037.706,334.220,-124.051,172.171,43.711,158.473
C07125=1037.717,334.585,-124.104,172.179,43.714,158.474
C07126=1037.728,334.951,-124.157,172.187,43.717,158.476
C07127=1037.739,335.317,-124.211,172.194,43.721,158.477
C07128=1037.746,335.564,-124.246,172.199,43.723,158.478
C07129=1037.753,335.811,-124.283,172.204,43.726,158.479
C07130=1037.761,336.059,-124.319,172.209,43.728,158.480
C07131=1037.768,336.306,-124.355,172.215,43.730,158.481
C07132=1037.775,336.553,-124.392,172.220,43.732,158.482
C07133=1037.782,336.801,-124.428,172.225,43.735,158.483
C07134=1037.789,337.047,-124.464,172.230,43.737,158.484
C07135=1037.797,337.295,-124.500,172.235,43.740,158.485
C07136=1037.805,337.542,-124.537,172.240,43.742,158.486
C07137=1037.812,337.790,-124.573,172.245,43.744,158.487
C07138=1037.819,338.037,-124.609,172.250,43.747,158.488
C07139=1037.827,338.284,-124.646,172.255,43.749,158.489
C07140=1037.834,338.531,-124.682,172.261,43.752,158.490
C07141=1037.842,338.779,-124.719,172.266,43.754,158.491
C07142=1037.849,339.026,-124.755,172.271,43.756,158.492
C07143=1037.856,339.273,-124.791,172.276,43.759,158.493
C07144=1037.864,339.520,-124.828,172.282,43.761,158.494
C07145=1037.872,339.767,-124.864,172.287,43.763,158.495
C07146=1037.879,340.015,-124.901,172.292,43.766,158.496
C07147=1037.886,340.261,-124.938,172.297,43.768,158.497
C07148=1037.894,340.509,-124.974,172.303,43.771,158.498
C07149=1037.902,340.756,-125.010,172.308,43.773,158.499
C07150=1037.909,341.003,-125.048,172.313,43.776,158.500
C07151=1037.916,341.251,-125.084,172.319,43.778,158.501
C07152=1037.924,341.498,-125.120,172.324,43.781,158.502
C07153=1037.931,341.745,-125.158,172.329,43.783,158.503
C07154=1037.939,341.993,-125.194,172.335,43.786,158.504
C07155=1037.946,342.239,-125.231,172.340,43.788,158.505
C07156=1037.953,342.487,-125.267,172.345,43.791,158.506
C07157=1037.961,342.734,-125.305,172.351,43.794,158.508
C07158=1037.969,342.981,-125.342,172.356,43.796,158.509
C07159=1037.975,343.228,-125.379,172.361,43.799,158.510
C07160=1037.983,343.475,-125.416,172.366,43.801,158.511
C07161=1037.990,343.723,-125.452,172.372,43.804,158.512
C07162=1037.998,343.970,-125.489,172.377,43.806,158.513
C07163=1038.006,344.217,-125.527,172.382,43.809,158.514
C07164=1038.014,344.464,-125.564,172.388,43.811,158.515
C07165=1038.021,344.711,-125.601,172.393,43.814,158.516
C07166=1038.029,344.958,-125.637,172.399,43.816,158.517
C07167=1038.036,345.205,-125.675,172.404,43.819,158.518
C07168=1038.044,345.452,-125.712,172.409,43.822,158.519
C07169=1038.051,345.700,-125.749,172.415,43.825,158.521
C07170=1038.058,345.947,-125.786,172.421,43.827,158.522
C07171=1038.066,346.194,-125.823,172.427,43.830,158.523
C07172=1038.073,346.441,-125.861,172.432,43.832,158.524
C07173=1038.081,346.688,-125.898,172.437,43.835,158.525
C07174=1038.088,346.935,-125.935,172.443,43.838,158.526
C07175=1038.096,347.182,-125.973,172.448,43.841,158.527
C07176=1038.104,347.429,-126.010,172.454,43.844,158.528
C07177=1038.111,347.676,-126.047,172.459,43.846,158.529
C07178=1038.119,347.924,-126.085,172.465,43.848,158.530
C07179=1038.127,348.171,-126.122,172.471,43.851,158.532
C07180=1038.137,348.533,-126.177,172.479,43.855,158.533
C07181=1038.149,348.895,-126.232,172.487,43.859,158.535
C07182=1038.160,349.256,-126.287,172.495,43.864,158.537
C07183=1038.171,349.619,-126.342,172.503,43.867,158.538
C07184=1038.178,349.866,-126.379,172.509,43.871,158.540
C07185=1038.186,350.113,-126.417,172.515,43.873,158.541
C07186=1038.194,350.360,-126.454,172.521,43.876,158.542
C07187=1038.202,350.607,-126.492,172.526,43.879,158.543
C07188=1038.209,350.854,-126.530,172.532,43.882,158.544
C07189=1038.217,351.101,-126.568,172.537,43.884,158.545
C07190=1038.224,351.348,-126.605,172.544,43.887,158.547
C07191=1038.232,351.595,-126.644,172.549,43.890,158.548
C07192=1038.240,351.842,-126.681,172.555,43.893,158.549
C07193=1038.248,352.089,-126.719,172.560,43.896,158.550
C07194=1038.255,352.337,-126.757,172.566,43.899,158.551
C07195=1038.263,352.583,-126.795,172.572,43.902,158.552
C07196=1038.270,352.830,-126.833,172.578,43.905,158.554
C07197=1038.278,353.077,-126.871,172.583,43.908,158.555
C07198=1038.286,353.325,-126.909,172.589,43.911,158.556
C07199=1038.293,353.571,-126.947,172.595,43.913,158.557
C07200=1038.302,353.818,-126.985,172.601,43.917,158.559
C07201=1038.309,354.065,-127.023,172.606,43.919,158.560
C07202=1038.317,354.312,-127.061,172.613,43.923,158.561
C07203=1038.325,354.559,-127.099,172.619,43.925,158.562
C07204=1038.332,354.806,-127.137,172.624,43.928,158.563
C07205=1038.340,355.053,-127.176,172.631,43.931,158.565
C07206=1038.348,355.300,-127.214,172.636,43.934,158.566
C07207=1038.355,355.547,-127.252,172.642,43.937,158.567
C07208=1038.363,355.794,-127.290,172.648,43.940,158.568
C07209=1038.371,356.041,-127.328,172.654,43.943,158.570
